MoveL Offs(p0,48.4696,297.2024, 0), v100, z5, tool0;
MoveL Offs(p0,48.6625,297.275, 0), v100, z5, tool0;
MoveL Offs(p0,48.848800000000004,297.9032, 0), v100, z5, tool0;
MoveL Offs(p0,48.7981,298.2614, 0), v100, z5, tool0;
MoveL Offs(p0,48.7,298.7, 0), v100, z5, tool0;
MoveL Offs(p0,48.48880000000001,299.4760000000001, 0), v100, z5, tool0;
MoveL Offs(p0,48.3652,299.978, 0), v100, z5, tool0;
MoveL Offs(p0,48.234399999999994,300.5400000000001, 0), v100, z5, tool0;
MoveL Offs(p0,48.1,301.15, 0), v100, z5, tool0;
MoveL Offs(p0,47.965599999999995,301.796, 0), v100, z5, tool0;
MoveL Offs(p0,47.834799999999994,302.466, 0), v100, z5, tool0;
MoveL Offs(p0,47.711200000000005,303.148, 0), v100, z5, tool0;
MoveL Offs(p0,47.598400000000005,303.83000000000004, 0), v100, z5, tool0;
MoveL Offs(p0,47.5,304.5, 0), v100, z5, tool0;
MoveL Offs(p0,47.17200000000001,306.3952000000001, 0), v100, z5, tool0;
MoveL Offs(p0,47.086,307.0218, 0), v100, z5, tool0;
MoveL Offs(p0,47.06000000000001,307.4456, 0), v100, z5, tool0;
MoveL Offs(p0,47.1,307.675, 0), v100, z5, tool0;
MoveL Offs(p0,47.211999999999996,307.7184, 0), v100, z5, tool0;
MoveL Offs(p0,48.040000000000006,306.8166, 0), v100, z5, tool0;
MoveL Offs(p0,48.5,306.2, 0), v100, z5, tool0;
MoveL Offs(p0,48.75480000000001,305.8350000000001, 0), v100, z5, tool0;
MoveL Offs(p0,48.97840000000001,305.46400000000006, 0), v100, z5, tool0;
MoveL Offs(p0,49.169599999999996,305.09299999999996, 0), v100, z5, tool0;
MoveL Offs(p0,49.3272,304.728, 0), v100, z5, tool0;
MoveL Offs(p0,49.45,304.375, 0), v100, z5, tool0;
MoveL Offs(p0,49.53680000000001,304.04, 0), v100, z5, tool0;
MoveL Offs(p0,49.586400000000005,303.729, 0), v100, z5, tool0;
MoveL Offs(p0,49.5976,303.44800000000004, 0), v100, z5, tool0;
MoveL Offs(p0,49.5692,303.20300000000003, 0), v100, z5, tool0;
MoveL Offs(p0,49.5,303.0, 0), v100, z5, tool0;
MoveL Offs(p0,49.5,303.0, 0), v100, z5, tool0;
MoveJ Offs(p0,394.7,303.0, 10), v100, z1, tool0;
MoveL Offs(p0,393.5853000000001,301.9654, 0), v100, z5, tool0;
MoveL Offs(p0,392.4784000000001,300.6392000000001, 0), v100, z5, tool0;
MoveL Offs(p0,391.4051,299.07779999999997, 0), v100, z5, tool0;
MoveL Offs(p0,390.3912,297.3376, 0), v100, z5, tool0;
MoveL Offs(p0,389.4625,295.475, 0), v100, z5, tool0;
MoveL Offs(p0,388.6448,293.5464, 0), v100, z5, tool0;
MoveL Offs(p0,387.9639,291.6082, 0), v100, z5, tool0;
MoveL Offs(p0,387.4456,289.71680000000003, 0), v100, z5, tool0;
MoveL Offs(p0,387.1157,287.9286, 0), v100, z5, tool0;
MoveL Offs(p0,387.0,286.3, 0), v100, z5, tool0;
MoveL Offs(p0,387.2152000000001,283.32400000000007, 0), v100, z5, tool0;
MoveL Offs(p0,387.4968,281.96200000000005, 0), v100, z5, tool0;
MoveL Offs(p0,387.90560000000005,280.65999999999997, 0), v100, z5, tool0;
MoveL Offs(p0,388.45,279.4, 0), v100, z5, tool0;
MoveL Offs(p0,389.1384,278.164, 0), v100, z5, tool0;
MoveL Offs(p0,389.9792,276.934, 0), v100, z5, tool0;
MoveL Offs(p0,390.9808,275.692, 0), v100, z5, tool0;
MoveL Offs(p0,392.15160000000003,274.42, 0), v100, z5, tool0;
MoveL Offs(p0,393.5,273.1, 0), v100, z5, tool0;
MoveL Offs(p0,394.37790000000007,272.2835000000001, 0), v100, z5, tool0;
MoveL Offs(p0,395.0992000000001,271.56000000000006, 0), v100, z5, tool0;
MoveL Offs(p0,395.6753,270.90849999999995, 0), v100, z5, tool0;
MoveL Offs(p0,396.11760000000004,270.30800000000005, 0), v100, z5, tool0;
MoveL Offs(p0,396.4375,269.7375, 0), v100, z5, tool0;
MoveL Offs(p0,396.64639999999997,269.176, 0), v100, z5, tool0;
MoveL Offs(p0,396.7557,268.6025, 0), v100, z5, tool0;
MoveL Offs(p0,396.77680000000004,267.996, 0), v100, z5, tool0;
MoveL Offs(p0,396.72110000000004,267.3355, 0), v100, z5, tool0;
MoveL Offs(p0,396.6,266.6, 0), v100, z5, tool0;
MoveL Offs(p0,396.2397,265.0522, 0), v100, z5, tool0;
MoveL Offs(p0,395.7936000000001,263.8056000000001, 0), v100, z5, tool0;
MoveL Offs(p0,395.1338999999999,262.8254, 0), v100, z5, tool0;
MoveL Offs(p0,394.13280000000003,262.0768, 0), v100, z5, tool0;
MoveL Offs(p0,392.6625,261.525, 0), v100, z5, tool0;
MoveL Offs(p0,390.59520000000003,261.1352, 0), v100, z5, tool0;
MoveL Offs(p0,387.8031,260.87260000000003, 0), v100, z5, tool0;
MoveL Offs(p0,384.1584,260.7024, 0), v100, z5, tool0;
MoveL Offs(p0,379.5333,260.5898, 0), v100, z5, tool0;
MoveL Offs(p0,373.8,260.5, 0), v100, z5, tool0;
MoveL Offs(p0,359.3056,260.172, 0), v100, z5, tool0;
MoveL Offs(p0,356.8625,260.0, 0), v100, z5, tool0;
MoveL Offs(p0,354.7344,259.78000000000003, 0), v100, z5, tool0;
MoveL Offs(p0,352.8427,259.506, 0), v100, z5, tool0;
MoveL Offs(p0,351.10880000000003,259.172, 0), v100, z5, tool0;
MoveL Offs(p0,349.45410000000004,258.77200000000005, 0), v100, z5, tool0;
MoveL Offs(p0,347.8,258.3, 0), v100, z5, tool0;
MoveL Offs(p0,346.68620000000004,257.98850000000004, 0), v100, z5, tool0;
MoveL Offs(p0,345.6336000000001,257.71600000000007, 0), v100, z5, tool0;
MoveL Offs(p0,344.6554,257.4855, 0), v100, z5, tool0;
MoveL Offs(p0,343.76480000000004,257.3, 0), v100, z5, tool0;
MoveL Offs(p0,342.975,257.1625, 0), v100, z5, tool0;
MoveL Offs(p0,342.2992,257.076, 0), v100, z5, tool0;
MoveL Offs(p0,341.7506,257.0435, 0), v100, z5, tool0;
MoveL Offs(p0,341.34240000000005,257.06800000000004, 0), v100, z5, tool0;
MoveL Offs(p0,341.0878,257.15250000000003, 0), v100, z5, tool0;
MoveL Offs(p0,341.0,257.3, 0), v100, z5, tool0;
MoveL Offs(p0,341.26160000000016,258.04080000000005, 0), v100, z5, tool0;
MoveL Offs(p0,341.57239999999996,258.7112, 0), v100, z5, tool0;
MoveL Offs(p0,341.9888,259.5544, 0), v100, z5, tool0;
MoveL Offs(p0,342.5,260.55, 0), v100, z5, tool0;
MoveL Offs(p0,343.0952,261.6776, 0), v100, z5, tool0;
MoveL Offs(p0,343.76359999999994,262.91679999999997, 0), v100, z5, tool0;
MoveL Offs(p0,344.49440000000004,264.2472000000001, 0), v100, z5, tool0;
MoveL Offs(p0,345.2768,265.64840000000004, 0), v100, z5, tool0;
MoveL Offs(p0,346.1,267.1, 0), v100, z5, tool0;
MoveL Offs(p0,347.2601000000001,269.11800000000005, 0), v100, z5, tool0;
MoveL Offs(p0,348.22880000000015,270.87200000000007, 0), v100, z5, tool0;
MoveL Offs(p0,349.0187,272.392, 0), v100, z5, tool0;
MoveL Offs(p0,349.64240000000007,273.70799999999997, 0), v100, z5, tool0;
MoveL Offs(p0,350.1125,274.85, 0), v100, z5, tool0;
MoveL Offs(p0,350.4416,275.848, 0), v100, z5, tool0;
MoveL Offs(p0,350.6423,276.732, 0), v100, z5, tool0;
MoveL Offs(p0,350.7272,277.53200000000004, 0), v100, z5, tool0;
MoveL Offs(p0,350.70889999999997,278.278, 0), v100, z5, tool0;
MoveL Offs(p0,350.6,279.0, 0), v100, z5, tool0;
MoveL Offs(p0,350.9,282.1, 0), v100, z5, tool0;
MoveL Offs(p0,351.32,282.6504, 0), v100, z5, tool0;
MoveL Offs(p0,351.902,283.2392, 0), v100, z5, tool0;
MoveL Offs(p0,352.66400000000004,283.8928, 0), v100, z5, tool0;
MoveL Offs(p0,353.62399999999997,284.63759999999996, 0), v100, z5, tool0;
MoveL Offs(p0,354.8,285.5, 0), v100, z5, tool0;
MoveL Offs(p0,356.8775,286.9497, 0), v100, z5, tool0;
MoveL Offs(p0,359.34800000000007,288.5176, 0), v100, z5, tool0;
MoveL Offs(p0,362.14849999999996,290.1719, 0), v100, z5, tool0;
MoveL Offs(p0,365.216,291.8808, 0), v100, z5, tool0;
MoveL Offs(p0,368.4875,293.6125, 0), v100, z5, tool0;
MoveL Offs(p0,371.9,295.3352, 0), v100, z5, tool0;
MoveL Offs(p0,375.3905,297.0171, 0), v100, z5, tool0;
MoveL Offs(p0,378.896,298.6264, 0), v100, z5, tool0;
MoveL Offs(p0,382.3535,300.1313, 0), v100, z5, tool0;
MoveL Offs(p0,385.7,301.5, 0), v100, z5, tool0;
MoveL Offs(p0,388.5062000000001,302.5680000000001, 0), v100, z5, tool0;
MoveL Offs(p0,390.8696000000001,303.4320000000001, 0), v100, z5, tool0;
MoveL Offs(p0,392.7974,304.092, 0), v100, z5, tool0;
MoveL Offs(p0,394.29679999999996,304.54800000000006, 0), v100, z5, tool0;
MoveL Offs(p0,395.375,304.8, 0), v100, z5, tool0;
MoveL Offs(p0,396.0392,304.84800000000007, 0), v100, z5, tool0;
MoveL Offs(p0,396.2966,304.692, 0), v100, z5, tool0;
MoveL Offs(p0,396.1544,304.332, 0), v100, z5, tool0;
MoveL Offs(p0,395.61980000000005,303.76800000000003, 0), v100, z5, tool0;
MoveL Offs(p0,394.7,303.0, 0), v100, z5, tool0;
MoveL Offs(p0,394.7,303.0, 0), v100, z5, tool0;
MoveJ Offs(p0,22.5,271.1, 10), v100, z1, tool0;
MoveL Offs(p0,23.33780000000001,268.8337, 0), v100, z5, tool0;
MoveL Offs(p0,24.18640000000001,266.6856000000001, 0), v100, z5, tool0;
MoveL Offs(p0,25.068599999999996,264.6119, 0), v100, z5, tool0;
MoveL Offs(p0,26.0072,262.5688, 0), v100, z5, tool0;
MoveL Offs(p0,27.025,260.5125, 0), v100, z5, tool0;
MoveL Offs(p0,28.144799999999996,258.39919999999995, 0), v100, z5, tool0;
MoveL Offs(p0,29.389400000000002,256.1851, 0), v100, z5, tool0;
MoveL Offs(p0,30.781600000000005,253.8264, 0), v100, z5, tool0;
MoveL Offs(p0,32.3442,251.2793, 0), v100, z5, tool0;
MoveL Offs(p0,34.1,248.5, 0), v100, z5, tool0;
MoveL Offs(p0,34.850500000000004,247.28090000000003, 0), v100, z5, tool0;
MoveL Offs(p0,35.48400000000001,246.19920000000008, 0), v100, z5, tool0;
MoveL Offs(p0,36.003499999999995,245.24829999999997, 0), v100, z5, tool0;
MoveL Offs(p0,36.412,244.42160000000004, 0), v100, z5, tool0;
MoveL Offs(p0,36.7125,243.7125, 0), v100, z5, tool0;
MoveL Offs(p0,36.908,243.1144, 0), v100, z5, tool0;
MoveL Offs(p0,37.0015,242.62070000000003, 0), v100, z5, tool0;
MoveL Offs(p0,36.996,242.22480000000004, 0), v100, z5, tool0;
MoveL Offs(p0,36.8945,241.9201, 0), v100, z5, tool0;
MoveL Offs(p0,36.7,241.7, 0), v100, z5, tool0;
MoveL Offs(p0,36.42160000000001,241.45840000000007, 0), v100, z5, tool0;
MoveL Offs(p0,36.3859,241.37959999999998, 0), v100, z5, tool0;
MoveL Offs(p0,36.41680000000001,241.3272, 0), v100, z5, tool0;
MoveL Offs(p0,37.17040000000001,241.3576, 0), v100, z5, tool0;
MoveL Offs(p0,37.5073,241.4192, 0), v100, z5, tool0;
MoveL Offs(p0,37.9,241.5, 0), v100, z5, tool0;
MoveL Offs(p0,38.72960000000001,241.7272000000001, 0), v100, z5, tool0;
MoveL Offs(p0,39.0484,241.7853, 0), v100, z5, tool0;
MoveL Offs(p0,39.30480000000001,241.8056, 0), v100, z5, tool0;
MoveL Offs(p0,39.5,241.7875, 0), v100, z5, tool0;
MoveL Offs(p0,39.635200000000005,241.7304, 0), v100, z5, tool0;
MoveL Offs(p0,39.6,241.1, 0), v100, z5, tool0;
MoveL Offs(p0,39.3993,240.57799999999997, 0), v100, z5, tool0;
MoveL Offs(p0,39.905100000000004,240.18200000000002, 0), v100, z5, tool0;
MoveL Offs(p0,40.1,240.2, 0), v100, z5, tool0;
MoveL Offs(p0,40.9136,239.93179999999998, 0), v100, z5, tool0;
MoveL Offs(p0,41.24720000000001,239.66559999999998, 0), v100, z5, tool0;
MoveL Offs(p0,41.6,239.325, 0), v100, z5, tool0;
MoveL Offs(p0,41.9648,238.91840000000002, 0), v100, z5, tool0;
MoveL Offs(p0,42.3344,238.4542, 0), v100, z5, tool0;
MoveL Offs(p0,42.701600000000006,237.94080000000002, 0), v100, z5, tool0;
MoveL Offs(p0,43.0592,237.3866, 0), v100, z5, tool0;
MoveL Offs(p0,43.4,236.8, 0), v100, z5, tool0;
MoveL Offs(p0,43.838300000000004,235.98240000000004, 0), v100, z5, tool0;
MoveL Offs(p0,44.19440000000001,235.2632000000001, 0), v100, z5, tool0;
MoveL Offs(p0,44.470099999999995,234.6328, 0), v100, z5, tool0;
MoveL Offs(p0,44.66720000000001,234.08160000000004, 0), v100, z5, tool0;
MoveL Offs(p0,44.7875,233.6, 0), v100, z5, tool0;
MoveL Offs(p0,44.832800000000006,233.17839999999995, 0), v100, z5, tool0;
MoveL Offs(p0,44.804899999999996,232.80720000000002, 0), v100, z5, tool0;
MoveL Offs(p0,44.705600000000004,232.4768, 0), v100, z5, tool0;
MoveL Offs(p0,44.5367,232.17759999999998, 0), v100, z5, tool0;
MoveL Offs(p0,44.3,231.9, 0), v100, z5, tool0;
MoveL Offs(p0,44.02900000000001,231.66020000000003, 0), v100, z5, tool0;
MoveL Offs(p0,43.75200000000001,231.48160000000007, 0), v100, z5, tool0;
MoveL Offs(p0,43.463,231.3654, 0), v100, z5, tool0;
MoveL Offs(p0,43.156000000000006,231.3128, 0), v100, z5, tool0;
MoveL Offs(p0,42.825,231.325, 0), v100, z5, tool0;
MoveL Offs(p0,42.464,231.40320000000003, 0), v100, z5, tool0;
MoveL Offs(p0,42.067,231.5486, 0), v100, z5, tool0;
MoveL Offs(p0,40.6,232.4, 0), v100, z5, tool0;
MoveL Offs(p0,40.16270000000001,232.67810000000003, 0), v100, z5, tool0;
MoveL Offs(p0,39.75360000000001,232.96880000000004, 0), v100, z5, tool0;
MoveL Offs(p0,39.37689999999999,233.2667, 0), v100, z5, tool0;
MoveL Offs(p0,39.0368,233.56640000000002, 0), v100, z5, tool0;
MoveL Offs(p0,38.7375,233.8625, 0), v100, z5, tool0;
MoveL Offs(p0,38.4832,234.14960000000002, 0), v100, z5, tool0;
MoveL Offs(p0,38.2781,234.4223, 0), v100, z5, tool0;
MoveL Offs(p0,38.126400000000004,234.67520000000005, 0), v100, z5, tool0;
MoveL Offs(p0,38.032300000000006,234.9029, 0), v100, z5, tool0;
MoveL Offs(p0,38.0,235.1, 0), v100, z5, tool0;
MoveL Offs(p0,37.751599999999996,235.95049999999998, 0), v100, z5, tool0;
MoveL Offs(p0,37.5712,236.348, 0), v100, z5, tool0;
MoveL Offs(p0,37.35,236.7875, 0), v100, z5, tool0;
MoveL Offs(p0,37.0928,237.26, 0), v100, z5, tool0;
MoveL Offs(p0,36.8044,237.75650000000002, 0), v100, z5, tool0;
MoveL Offs(p0,36.48960000000001,238.26800000000003, 0), v100, z5, tool0;
MoveL Offs(p0,36.153200000000005,238.78550000000004, 0), v100, z5, tool0;
MoveL Offs(p0,35.8,239.3, 0), v100, z5, tool0;
MoveL Offs(p0,34.16930000000001,241.69430000000006, 0), v100, z5, tool0;
MoveL Offs(p0,32.39040000000001,244.57040000000006, 0), v100, z5, tool0;
MoveL Offs(p0,30.5431,247.7681, 0), v100, z5, tool0;
MoveL Offs(p0,28.7072,251.12720000000004, 0), v100, z5, tool0;
MoveL Offs(p0,26.9625,254.4875, 0), v100, z5, tool0;
MoveL Offs(p0,25.388799999999996,257.6888, 0), v100, z5, tool0;
MoveL Offs(p0,24.0659,260.5709, 0), v100, z5, tool0;
MoveL Offs(p0,23.073600000000003,262.9736, 0), v100, z5, tool0;
MoveL Offs(p0,22.4917,264.73670000000004, 0), v100, z5, tool0;
MoveL Offs(p0,22.4,265.7, 0), v100, z5, tool0;
MoveL Offs(p0,22.2,267.0, 0), v100, z5, tool0;
MoveL Offs(p0,21.6107,267.5379, 0), v100, z5, tool0;
MoveL Offs(p0,20.89360000000001,269.02320000000003, 0), v100, z5, tool0;
MoveL Offs(p0,20.094900000000003,271.26329999999996, 0), v100, z5, tool0;
MoveL Offs(p0,19.2608,274.0656, 0), v100, z5, tool0;
MoveL Offs(p0,18.4375,277.2375, 0), v100, z5, tool0;
MoveL Offs(p0,17.6712,280.5864, 0), v100, z5, tool0;
MoveL Offs(p0,17.0081,283.9197, 0), v100, z5, tool0;
MoveL Offs(p0,16.494400000000002,287.0448, 0), v100, z5, tool0;
MoveL Offs(p0,16.1763,289.76910000000004, 0), v100, z5, tool0;
MoveL Offs(p0,16.1,291.9, 0), v100, z5, tool0;
MoveL Offs(p0,16.3214,292.1826, 0), v100, z5, tool0;
MoveL Offs(p0,16.675,291.375, 0), v100, z5, tool0;
MoveL Offs(p0,16.8992,290.7048, 0), v100, z5, tool0;
MoveL Offs(p0,17.1486,289.8714, 0), v100, z5, tool0;
MoveL Offs(p0,17.418400000000002,288.8856, 0), v100, z5, tool0;
MoveL Offs(p0,17.7038,287.75820000000004, 0), v100, z5, tool0;
MoveL Offs(p0,18.0,286.5, 0), v100, z5, tool0;
MoveL Offs(p0,18.328500000000005,285.11030000000005, 0), v100, z5, tool0;
MoveL Offs(p0,18.708000000000006,283.6024000000001, 0), v100, z5, tool0;
MoveL Offs(p0,19.1295,282.00809999999996, 0), v100, z5, tool0;
MoveL Offs(p0,19.584,280.3592, 0), v100, z5, tool0;
MoveL Offs(p0,20.0625,278.6875, 0), v100, z5, tool0;
MoveL Offs(p0,20.556,277.02479999999997, 0), v100, z5, tool0;
MoveL Offs(p0,21.055500000000002,275.4029, 0), v100, z5, tool0;
MoveL Offs(p0,21.552000000000003,273.85360000000003, 0), v100, z5, tool0;
MoveL Offs(p0,22.0365,272.4087, 0), v100, z5, tool0;
MoveL Offs(p0,22.5,271.1, 0), v100, z5, tool0;
MoveL Offs(p0,22.5,271.1, 0), v100, z5, tool0;
MoveJ Offs(p0,36.1,288.1, 10), v100, z1, tool0;
MoveL Offs(p0,36.39620000000001,288.49760000000003, 0), v100, z5, tool0;
MoveL Offs(p0,36.68160000000002,288.9048000000001, 0), v100, z5, tool0;
MoveL Offs(p0,36.95139999999999,289.3132, 0), v100, z5, tool0;
MoveL Offs(p0,37.2008,289.71439999999996, 0), v100, z5, tool0;
MoveL Offs(p0,37.425,290.1, 0), v100, z5, tool0;
MoveL Offs(p0,37.6192,290.4616, 0), v100, z5, tool0;
MoveL Offs(p0,37.7786,290.7908, 0), v100, z5, tool0;
MoveL Offs(p0,37.8984,291.0792, 0), v100, z5, tool0;
MoveL Offs(p0,37.973800000000004,291.3184, 0), v100, z5, tool0;
MoveL Offs(p0,38.0,291.5, 0), v100, z5, tool0;
MoveL Offs(p0,38.6875,291.0625, 0), v100, z5, tool0;
MoveL Offs(p0,38.93599999999999,290.70079999999996, 0), v100, z5, tool0;
MoveL Offs(p0,39.2145,290.2659, 0), v100, z5, tool0;
MoveL Offs(p0,39.52,289.7656, 0), v100, z5, tool0;
MoveL Offs(p0,39.8495,289.20770000000005, 0), v100, z5, tool0;
MoveL Offs(p0,40.2,288.6, 0), v100, z5, tool0;
MoveL Offs(p0,42.2,284.6, 0), v100, z5, tool0;
MoveL Offs(p0,44.0,286.9, 0), v100, z5, tool0;
MoveL Offs(p0,44.4371,287.49449999999996, 0), v100, z5, tool0;
MoveL Offs(p0,44.79680000000001,287.9600000000001, 0), v100, z5, tool0;
MoveL Offs(p0,45.0917,288.29949999999997, 0), v100, z5, tool0;
MoveL Offs(p0,45.3344,288.516, 0), v100, z5, tool0;
MoveL Offs(p0,45.5375,288.6125, 0), v100, z5, tool0;
MoveL Offs(p0,45.7136,288.592, 0), v100, z5, tool0;
MoveL Offs(p0,45.8753,288.4575, 0), v100, z5, tool0;
MoveL Offs(p0,46.03520000000001,288.212, 0), v100, z5, tool0;
MoveL Offs(p0,46.2059,287.8585, 0), v100, z5, tool0;
MoveL Offs(p0,46.4,287.4, 0), v100, z5, tool0;
MoveL Offs(p0,46.998400000000004,284.9322, 0), v100, z5, tool0;
MoveL Offs(p0,47.41920000000002,281.10960000000006, 0), v100, z5, tool0;
MoveL Offs(p0,47.6708,276.2634, 0), v100, z5, tool0;
MoveL Offs(p0,47.7616,270.7248, 0), v100, z5, tool0;
MoveL Offs(p0,47.7,264.825, 0), v100, z5, tool0;
MoveL Offs(p0,47.4944,258.89520000000005, 0), v100, z5, tool0;
MoveL Offs(p0,47.1532,253.2666, 0), v100, z5, tool0;
MoveL Offs(p0,46.68480000000001,248.27040000000002, 0), v100, z5, tool0;
MoveL Offs(p0,46.0976,244.23780000000002, 0), v100, z5, tool0;
MoveL Offs(p0,45.4,241.5, 0), v100, z5, tool0;
MoveL Offs(p0,44.52810000000001,240.81270000000004, 0), v100, z5, tool0;
MoveL Offs(p0,41.1367,243.1029, 0), v100, z5, tool0;
MoveL Offs(p0,38.8464,245.75280000000004, 0), v100, z5, tool0;
MoveL Offs(p0,36.3125,249.1875, 0), v100, z5, tool0;
MoveL Offs(p0,33.6496,253.24319999999997, 0), v100, z5, tool0;
MoveL Offs(p0,30.972299999999997,257.7561, 0), v100, z5, tool0;
MoveL Offs(p0,28.3952,262.5624, 0), v100, z5, tool0;
MoveL Offs(p0,26.0329,267.49830000000003, 0), v100, z5, tool0;
MoveL Offs(p0,24.0,272.4, 0), v100, z5, tool0;
MoveL Offs(p0,23.035600000000002,275.0069000000001, 0), v100, z5, tool0;
MoveL Offs(p0,22.188800000000004,277.5712000000001, 0), v100, z5, tool0;
MoveL Offs(p0,21.4692,280.0383, 0), v100, z5, tool0;
MoveL Offs(p0,20.886400000000002,282.3536, 0), v100, z5, tool0;
MoveL Offs(p0,20.45,284.4625, 0), v100, z5, tool0;
MoveL Offs(p0,20.1696,286.3104, 0), v100, z5, tool0;
MoveL Offs(p0,20.0548,287.84270000000004, 0), v100, z5, tool0;
MoveL Offs(p0,20.115200000000005,289.00480000000005, 0), v100, z5, tool0;
MoveL Offs(p0,20.3604,289.74210000000005, 0), v100, z5, tool0;
MoveL Offs(p0,20.8,290.0, 0), v100, z5, tool0;
MoveL Offs(p0,21.5047,289.703, 0), v100, z5, tool0;
MoveL Offs(p0,21.7984,289.48800000000006, 0), v100, z5, tool0;
MoveL Offs(p0,22.1125,289.225, 0), v100, z5, tool0;
MoveL Offs(p0,22.4416,288.91999999999996, 0), v100, z5, tool0;
MoveL Offs(p0,22.7803,288.579, 0), v100, z5, tool0;
MoveL Offs(p0,23.123200000000004,288.20799999999997, 0), v100, z5, tool0;
MoveL Offs(p0,23.4649,287.813, 0), v100, z5, tool0;
MoveL Offs(p0,23.8,287.4, 0), v100, z5, tool0;
MoveL Offs(p0,25.7,284.7, 0), v100, z5, tool0;
MoveL Offs(p0,28.0,288.4, 0), v100, z5, tool0;
MoveL Offs(p0,30.2,292.1, 0), v100, z5, tool0;
MoveL Offs(p0,32.2,288.9, 0), v100, z5, tool0;
MoveL Offs(p0,34.2,285.6, 0), v100, z5, tool0;
MoveL Offs(p0,36.1,288.1, 0), v100, z5, tool0;
MoveL Offs(p0,36.1,288.1, 0), v100, z5, tool0;
MoveJ Offs(p0,86.6,282.4, 10), v100, z1, tool0;
MoveL Offs(p0,86.38880000000003,279.65520000000004, 0), v100, z5, tool0;
MoveL Offs(p0,86.26520000000001,278.3698, 0), v100, z5, tool0;
MoveL Offs(p0,86.13440000000001,277.1696, 0), v100, z5, tool0;
MoveL Offs(p0,86.0,276.075, 0), v100, z5, tool0;
MoveL Offs(p0,85.8656,275.1064, 0), v100, z5, tool0;
MoveL Offs(p0,85.73479999999999,274.28419999999994, 0), v100, z5, tool0;
MoveL Offs(p0,85.61120000000001,273.62880000000007, 0), v100, z5, tool0;
MoveL Offs(p0,85.49839999999999,273.16060000000004, 0), v100, z5, tool0;
MoveL Offs(p0,85.4,272.9, 0), v100, z5, tool0;
MoveL Offs(p0,85.0895,272.0855, 0), v100, z5, tool0;
MoveL Offs(p0,84.976,271.676, 0), v100, z5, tool0;
MoveL Offs(p0,84.8625,271.2125, 0), v100, z5, tool0;
MoveL Offs(p0,84.752,270.70399999999995, 0), v100, z5, tool0;
MoveL Offs(p0,84.64750000000001,270.1595, 0), v100, z5, tool0;
MoveL Offs(p0,84.552,269.588, 0), v100, z5, tool0;
MoveL Offs(p0,84.4685,268.99850000000004, 0), v100, z5, tool0;
MoveL Offs(p0,84.4,268.4, 0), v100, z5, tool0;
MoveL Offs(p0,83.85910000000001,265.5085, 0), v100, z5, tool0;
MoveL Offs(p0,82.94080000000002,262.04400000000004, 0), v100, z5, tool0;
MoveL Offs(p0,81.71169999999998,258.1715, 0), v100, z5, tool0;
MoveL Offs(p0,80.2384,254.05599999999998, 0), v100, z5, tool0;
MoveL Offs(p0,78.5875,249.8625, 0), v100, z5, tool0;
MoveL Offs(p0,76.8256,245.756, 0), v100, z5, tool0;
MoveL Offs(p0,75.0193,241.9015, 0), v100, z5, tool0;
MoveL Offs(p0,73.2352,238.46400000000003, 0), v100, z5, tool0;
MoveL Offs(p0,71.5399,235.6085, 0), v100, z5, tool0;
MoveL Offs(p0,70.0,233.5, 0), v100, z5, tool0;
MoveL Offs(p0,69.5334,232.9835, 0), v100, z5, tool0;
MoveL Offs(p0,69.03920000000002,232.40400000000008, 0), v100, z5, tool0;
MoveL Offs(p0,68.52579999999999,231.7765, 0), v100, z5, tool0;
MoveL Offs(p0,68.00160000000001,231.11600000000004, 0), v100, z5, tool0;
MoveL Offs(p0,67.475,230.4375, 0), v100, z5, tool0;
MoveL Offs(p0,66.95439999999999,229.756, 0), v100, z5, tool0;
MoveL Offs(p0,66.4482,229.08649999999997, 0), v100, z5, tool0;
MoveL Offs(p0,65.9648,228.44400000000005, 0), v100, z5, tool0;
MoveL Offs(p0,65.51259999999999,227.84350000000003, 0), v100, z5, tool0;
MoveL Offs(p0,65.1,227.3, 0), v100, z5, tool0;
MoveL Offs(p0,64.72650000000002,226.77020000000002, 0), v100, z5, tool0;
MoveL Offs(p0,64.33200000000001,226.2656000000001, 0), v100, z5, tool0;
MoveL Offs(p0,63.9255,225.79339999999996, 0), v100, z5, tool0;
MoveL Offs(p0,63.516000000000005,225.3608, 0), v100, z5, tool0;
MoveL Offs(p0,63.1125,224.975, 0), v100, z5, tool0;
MoveL Offs(p0,62.724000000000004,224.64319999999998, 0), v100, z5, tool0;
MoveL Offs(p0,62.359500000000004,224.3726, 0), v100, z5, tool0;
MoveL Offs(p0,62.028,224.17040000000003, 0), v100, z5, tool0;
MoveL Offs(p0,61.7385,224.0438, 0), v100, z5, tool0;
MoveL Offs(p0,61.5,224.0, 0), v100, z5, tool0;
MoveL Offs(p0,60.981700000000004,224.25660000000002, 0), v100, z5, tool0;
MoveL Offs(p0,60.78560000000001,224.97280000000006, 0), v100, z5, tool0;
MoveL Offs(p0,60.8799,226.0682, 0), v100, z5, tool0;
MoveL Offs(p0,61.23280000000001,227.46239999999997, 0), v100, z5, tool0;
MoveL Offs(p0,61.8125,229.075, 0), v100, z5, tool0;
MoveL Offs(p0,62.58720000000001,230.82559999999998, 0), v100, z5, tool0;
MoveL Offs(p0,63.525099999999995,232.6338, 0), v100, z5, tool0;
MoveL Offs(p0,64.59440000000001,234.4192, 0), v100, z5, tool0;
MoveL Offs(p0,65.7633,236.1014, 0), v100, z5, tool0;
MoveL Offs(p0,67.0,237.6, 0), v100, z5, tool0;
MoveL Offs(p0,67.62470000000002,238.30800000000005, 0), v100, z5, tool0;
MoveL Offs(p0,68.28960000000002,239.10000000000014, 0), v100, z5, tool0;
MoveL Offs(p0,68.98089999999999,239.958, 0), v100, z5, tool0;
MoveL Offs(p0,69.68480000000001,240.86400000000003, 0), v100, z5, tool0;
MoveL Offs(p0,70.3875,241.8, 0), v100, z5, tool0;
MoveL Offs(p0,71.0752,242.74799999999996, 0), v100, z5, tool0;
MoveL Offs(p0,71.7341,243.69, 0), v100, z5, tool0;
MoveL Offs(p0,72.35040000000001,244.608, 0), v100, z5, tool0;
MoveL Offs(p0,72.91029999999999,245.484, 0), v100, z5, tool0;
MoveL Offs(p0,73.4,246.3, 0), v100, z5, tool0;
MoveL Offs(p0,74.3298,247.97310000000007, 0), v100, z5, tool0;
MoveL Offs(p0,75.45040000000003,250.1808000000001, 0), v100, z5, tool0;
MoveL Offs(p0,76.6886,252.7557, 0), v100, z5, tool0;
MoveL Offs(p0,77.9712,255.53040000000001, 0), v100, z5, tool0;
MoveL Offs(p0,79.225,258.3375, 0), v100, z5, tool0;
MoveL Offs(p0,80.3768,261.0096, 0), v100, z5, tool0;
MoveL Offs(p0,81.35340000000001,263.37929999999994, 0), v100, z5, tool0;
MoveL Offs(p0,82.08160000000001,265.27920000000006, 0), v100, z5, tool0;
MoveL Offs(p0,82.4882,266.54190000000006, 0), v100, z5, tool0;
MoveL Offs(p0,82.5,267.0, 0), v100, z5, tool0;
MoveL Offs(p0,82.7121,268.7934, 0), v100, z5, tool0;
MoveL Offs(p0,82.8264,269.2656, 0), v100, z5, tool0;
MoveL Offs(p0,82.95630000000001,269.77020000000005, 0), v100, z5, tool0;
MoveL Offs(p0,83.1,270.3, 0), v100, z5, tool0;
MoveL Offs(p0,83.40750000000001,271.3081, 0), v100, z5, tool0;
MoveL Offs(p0,83.67600000000002,272.26880000000006, 0), v100, z5, tool0;
MoveL Offs(p0,83.9145,273.23670000000004, 0), v100, z5, tool0;
MoveL Offs(p0,84.132,274.2664, 0), v100, z5, tool0;
MoveL Offs(p0,84.3375,275.4125, 0), v100, z5, tool0;
MoveL Offs(p0,84.53999999999999,276.7296, 0), v100, z5, tool0;
MoveL Offs(p0,84.74849999999999,278.2723, 0), v100, z5, tool0;
MoveL Offs(p0,84.97200000000001,280.09520000000003, 0), v100, z5, tool0;
MoveL Offs(p0,85.21950000000001,282.25290000000007, 0), v100, z5, tool0;
MoveL Offs(p0,85.5,284.8, 0), v100, z5, tool0;
MoveL Offs(p0,85.8197,287.23570000000007, 0), v100, z5, tool0;
MoveL Offs(p0,86.11360000000002,289.0336000000001, 0), v100, z5, tool0;
MoveL Offs(p0,86.3739,290.20989999999995, 0), v100, z5, tool0;
MoveL Offs(p0,86.5928,290.7808, 0), v100, z5, tool0;
MoveL Offs(p0,86.7625,290.7625, 0), v100, z5, tool0;
MoveL Offs(p0,86.87519999999999,290.1712, 0), v100, z5, tool0;
MoveL Offs(p0,86.9231,289.0231, 0), v100, z5, tool0;
MoveL Offs(p0,86.89840000000001,287.3344, 0), v100, z5, tool0;
MoveL Offs(p0,86.7933,285.1213, 0), v100, z5, tool0;
MoveL Offs(p0,86.6,282.4, 0), v100, z5, tool0;
MoveL Offs(p0,86.6,282.4, 0), v100, z5, tool0;
MoveJ Offs(p0,149.5,287.9, 10), v100, z1, tool0;
MoveL Offs(p0,149.73039999999997,286.9244, 0), v100, z5, tool0;
MoveL Offs(p0,149.7528,286.58480000000003, 0), v100, z5, tool0;
MoveL Offs(p0,149.75,286.25, 0), v100, z5, tool0;
MoveL Offs(p0,149.7232,285.92719999999997, 0), v100, z5, tool0;
MoveL Offs(p0,149.1777,284.40770000000003, 0), v100, z5, tool0;
MoveL Offs(p0,149.1664,284.30640000000005, 0), v100, z5, tool0;
MoveL Offs(p0,149.1875,284.2375, 0), v100, z5, tool0;
MoveL Offs(p0,149.60790000000003,284.2979, 0), v100, z5, tool0;
MoveL Offs(p0,149.8,284.4, 0), v100, z5, tool0;
MoveL Offs(p0,150.95559999999998,284.1885, 0), v100, z5, tool0;
MoveL Offs(p0,151.1312,283.656, 0), v100, z5, tool0;
MoveL Offs(p0,151.2,282.9375, 0), v100, z5, tool0;
MoveL Offs(p0,151.16079999999997,282.06000000000006, 0), v100, z5, tool0;
MoveL Offs(p0,151.0124,281.0505, 0), v100, z5, tool0;
MoveL Offs(p0,150.7536,279.93600000000004, 0), v100, z5, tool0;
MoveL Offs(p0,150.38320000000002,278.74350000000004, 0), v100, z5, tool0;
MoveL Offs(p0,148.91250000000005,274.55550000000005, 0), v100, z5, tool0;
MoveL Offs(p0,148.16800000000003,270.98400000000004, 0), v100, z5, tool0;
MoveL Offs(p0,147.6635,266.9385, 0), v100, z5, tool0;
MoveL Offs(p0,147.39600000000002,262.572, 0), v100, z5, tool0;
MoveL Offs(p0,147.3625,258.0375, 0), v100, z5, tool0;
MoveL Offs(p0,147.56,253.488, 0), v100, z5, tool0;
MoveL Offs(p0,147.9855,249.07649999999998, 0), v100, z5, tool0;
MoveL Offs(p0,148.63600000000002,244.95600000000005, 0), v100, z5, tool0;
MoveL Offs(p0,149.5085,241.2795, 0), v100, z5, tool0;
MoveL Offs(p0,150.6,238.2, 0), v100, z5, tool0;
MoveL Offs(p0,150.88770000000002,237.59880000000004, 0), v100, z5, tool0;
MoveL Offs(p0,151.14960000000002,237.00240000000002, 0), v100, z5, tool0;
MoveL Offs(p0,151.3839,236.42160000000004, 0), v100, z5, tool0;
MoveL Offs(p0,151.58880000000002,235.86720000000005, 0), v100, z5, tool0;
MoveL Offs(p0,151.7625,235.35, 0), v100, z5, tool0;
MoveL Offs(p0,151.90320000000003,234.8808, 0), v100, z5, tool0;
MoveL Offs(p0,152.0091,234.4704, 0), v100, z5, tool0;
MoveL Offs(p0,152.07840000000002,234.12960000000004, 0), v100, z5, tool0;
MoveL Offs(p0,152.10930000000002,233.8692, 0), v100, z5, tool0;
MoveL Offs(p0,152.1,233.7, 0), v100, z5, tool0;
MoveL Offs(p0,152.3952,233.2536, 0), v100, z5, tool0;
MoveL Offs(p0,152.5221,233.2723, 0), v100, z5, tool0;
MoveL Offs(p0,152.6664,233.3192, 0), v100, z5, tool0;
MoveL Offs(p0,152.8263,233.3949, 0), v100, z5, tool0;
MoveL Offs(p0,153.0,233.5, 0), v100, z5, tool0;
MoveL Offs(p0,153.9855,233.26510000000002, 0), v100, z5, tool0;
MoveL Offs(p0,154.0,233.1, 0), v100, z5, tool0;
MoveL Offs(p0,153.79520000000002,232.78000000000006, 0), v100, z5, tool0;
MoveL Offs(p0,153.55180000000001,232.60950000000003, 0), v100, z5, tool0;
MoveL Offs(p0,153.22560000000001,232.43599999999998, 0), v100, z5, tool0;
MoveL Offs(p0,152.825,232.2625, 0), v100, z5, tool0;
MoveL Offs(p0,152.35840000000002,232.092, 0), v100, z5, tool0;
MoveL Offs(p0,151.8342,231.9275, 0), v100, z5, tool0;
MoveL Offs(p0,151.26080000000002,231.77200000000002, 0), v100, z5, tool0;
MoveL Offs(p0,150.6466,231.62849999999997, 0), v100, z5, tool0;
MoveL Offs(p0,150.0,231.5, 0), v100, z5, tool0;
MoveL Offs(p0,148.71520000000004,231.22800000000007, 0), v100, z5, tool0;
MoveL Offs(p0,148.1118,231.0725, 0), v100, z5, tool0;
MoveL Offs(p0,147.5456,230.90800000000004, 0), v100, z5, tool0;
MoveL Offs(p0,147.025,230.7375, 0), v100, z5, tool0;
MoveL Offs(p0,146.55839999999998,230.564, 0), v100, z5, tool0;
MoveL Offs(p0,146.1542,230.39049999999997, 0), v100, z5, tool0;
MoveL Offs(p0,145.82080000000002,230.21999999999997, 0), v100, z5, tool0;
MoveL Offs(p0,145.56660000000002,230.05550000000002, 0), v100, z5, tool0;
MoveL Offs(p0,145.4,229.9, 0), v100, z5, tool0;
MoveL Offs(p0,145.04210000000003,229.44020000000006, 0), v100, z5, tool0;
MoveL Offs(p0,144.63680000000005,229.13760000000002, 0), v100, z5, tool0;
MoveL Offs(p0,144.19670000000002,228.98740000000004, 0), v100, z5, tool0;
MoveL Offs(p0,143.7344,228.9848, 0), v100, z5, tool0;
MoveL Offs(p0,143.2625,229.125, 0), v100, z5, tool0;
MoveL Offs(p0,142.7936,229.40319999999997, 0), v100, z5, tool0;
MoveL Offs(p0,141.9152,230.3544, 0), v100, z5, tool0;
MoveL Offs(p0,141.53090000000003,231.0178, 0), v100, z5, tool0;
MoveL Offs(p0,141.2,231.8, 0), v100, z5, tool0;
MoveL Offs(p0,139.91450000000003,236.19530000000003, 0), v100, z5, tool0;
MoveL Offs(p0,138.99200000000002,241.48640000000006, 0), v100, z5, tool0;
MoveL Offs(p0,138.4235,247.44109999999995, 0), v100, z5, tool0;
MoveL Offs(p0,138.2,253.8272, 0), v100, z5, tool0;
MoveL Offs(p0,138.3125,260.4125, 0), v100, z5, tool0;
MoveL Offs(p0,138.752,266.9648, 0), v100, z5, tool0;
MoveL Offs(p0,139.5095,273.25190000000003, 0), v100, z5, tool0;
MoveL Offs(p0,140.57600000000002,279.0416, 0), v100, z5, tool0;
MoveL Offs(p0,141.9425,284.1017, 0), v100, z5, tool0;
MoveL Offs(p0,143.6,288.2, 0), v100, z5, tool0;
MoveL Offs(p0,144.127,289.007, 0), v100, z5, tool0;
MoveL Offs(p0,144.73200000000003,289.62800000000004, 0), v100, z5, tool0;
MoveL Offs(p0,145.391,290.063, 0), v100, z5, tool0;
MoveL Offs(p0,146.08,290.312, 0), v100, z5, tool0;
MoveL Offs(p0,146.775,290.375, 0), v100, z5, tool0;
MoveL Offs(p0,147.452,290.25199999999995, 0), v100, z5, tool0;
MoveL Offs(p0,148.087,289.943, 0), v100, z5, tool0;
MoveL Offs(p0,148.656,289.44800000000004, 0), v100, z5, tool0;
MoveL Offs(p0,149.13500000000002,288.767, 0), v100, z5, tool0;
MoveL Offs(p0,149.5,287.9, 0), v100, z5, tool0;
MoveL Offs(p0,149.5,287.9, 0), v100, z5, tool0;
MoveJ Offs(p0,156.2,285.7, 10), v100, z1, tool0;
MoveL Offs(p0,156.5645,282.5032, 0), v100, z5, tool0;
MoveL Offs(p0,156.96,281.3624, 0), v100, z5, tool0;
MoveL Offs(p0,157.4875,280.2, 0), v100, z5, tool0;
MoveL Offs(p0,158.144,279.0256, 0), v100, z5, tool0;
MoveL Offs(p0,158.92649999999998,277.84880000000004, 0), v100, z5, tool0;
MoveL Offs(p0,159.83200000000002,276.67920000000004, 0), v100, z5, tool0;
MoveL Offs(p0,160.85750000000002,275.5264, 0), v100, z5, tool0;
MoveL Offs(p0,162.0,274.4, 0), v100, z5, tool0;
MoveL Offs(p0,162.92490000000004,273.48810000000003, 0), v100, z5, tool0;
MoveL Offs(p0,163.66320000000005,272.72080000000005, 0), v100, z5, tool0;
MoveL Offs(p0,164.2203,272.0806999999999, 0), v100, z5, tool0;
MoveL Offs(p0,164.60160000000002,271.5504, 0), v100, z5, tool0;
MoveL Offs(p0,164.8125,271.1125, 0), v100, z5, tool0;
MoveL Offs(p0,164.8584,270.7496, 0), v100, z5, tool0;
MoveL Offs(p0,164.74470000000002,270.4443, 0), v100, z5, tool0;
MoveL Offs(p0,164.4768,270.17920000000004, 0), v100, z5, tool0;
MoveL Offs(p0,164.0601,269.93690000000004, 0), v100, z5, tool0;
MoveL Offs(p0,163.5,269.7, 0), v100, z5, tool0;
MoveL Offs(p0,161.76479999999998,270.26969999999994, 0), v100, z5, tool0;
MoveL Offs(p0,161.0616,270.8584, 0), v100, z5, tool0;
MoveL Offs(p0,160.35,271.5875, 0), v100, z5, tool0;
MoveL Offs(p0,159.6624,272.4216, 0), v100, z5, tool0;
MoveL Offs(p0,159.03119999999998,273.32529999999997, 0), v100, z5, tool0;
MoveL Offs(p0,158.4888,274.2632, 0), v100, z5, tool0;
MoveL Offs(p0,158.0676,275.19989999999996, 0), v100, z5, tool0;
MoveL Offs(p0,157.8,276.1, 0), v100, z5, tool0;
MoveL Offs(p0,157.57410000000002,276.80649999999997, 0), v100, z5, tool0;
MoveL Offs(p0,157.4832,277.02799999999996, 0), v100, z5, tool0;
MoveL Offs(p0,157.3875,277.2375, 0), v100, z5, tool0;
MoveL Offs(p0,157.2888,277.43199999999996, 0), v100, z5, tool0;
MoveL Offs(p0,157.1889,277.6085, 0), v100, z5, tool0;
MoveL Offs(p0,157.08960000000002,277.764, 0), v100, z5, tool0;
MoveL Offs(p0,156.9927,277.8955, 0), v100, z5, tool0;
MoveL Offs(p0,156.9,278.0, 0), v100, z5, tool0;
MoveL Offs(p0,156.6207,278.41780000000006, 0), v100, z5, tool0;
MoveL Offs(p0,156.22560000000004,279.1944000000001, 0), v100, z5, tool0;
MoveL Offs(p0,155.7489,280.2446, 0), v100, z5, tool0;
MoveL Offs(p0,155.22480000000002,281.4832, 0), v100, z5, tool0;
MoveL Offs(p0,154.6875,282.825, 0), v100, z5, tool0;
MoveL Offs(p0,154.17120000000003,284.1848, 0), v100, z5, tool0;
MoveL Offs(p0,153.71009999999998,285.47740000000005, 0), v100, z5, tool0;
MoveL Offs(p0,153.3384,286.61760000000004, 0), v100, z5, tool0;
MoveL Offs(p0,153.0903,287.52020000000005, 0), v100, z5, tool0;
MoveL Offs(p0,153.0,288.1, 0), v100, z5, tool0;
MoveL Offs(p0,153.34560000000002,288.6632, 0), v100, z5, tool0;
MoveL Offs(p0,153.525,288.75, 0), v100, z5, tool0;
MoveL Offs(p0,153.7344,288.81280000000004, 0), v100, z5, tool0;
MoveL Offs(p0,153.97020000000003,288.8504, 0), v100, z5, tool0;
MoveL Offs(p0,154.2288,288.8616, 0), v100, z5, tool0;
MoveL Offs(p0,154.5066,288.84520000000003, 0), v100, z5, tool0;
MoveL Offs(p0,154.8,288.8, 0), v100, z5, tool0;
MoveL Offs(p0,155.42560000000006,288.5448000000001, 0), v100, z5, tool0;
MoveL Offs(p0,155.6694,288.35720000000003, 0), v100, z5, tool0;
MoveL Offs(p0,155.86880000000002,288.1264, 0), v100, z5, tool0;
MoveL Offs(p0,156.025,287.85, 0), v100, z5, tool0;
MoveL Offs(p0,156.1392,287.52560000000005, 0), v100, z5, tool0;
MoveL Offs(p0,156.2126,287.1508, 0), v100, z5, tool0;
MoveL Offs(p0,156.2464,286.7232, 0), v100, z5, tool0;
MoveL Offs(p0,156.2418,286.2404, 0), v100, z5, tool0;
MoveL Offs(p0,156.2,285.7, 0), v100, z5, tool0;
MoveL Offs(p0,156.2,285.7, 0), v100, z5, tool0;
MoveJ Offs(p0,172.8,284.9, 10), v100, z1, tool0;
MoveL Offs(p0,173.7997,284.68750000000006, 0), v100, z5, tool0;
MoveL Offs(p0,174.74960000000004,284.4720000000001, 0), v100, z5, tool0;
MoveL Offs(p0,175.63590000000002,284.2565, 0), v100, z5, tool0;
MoveL Offs(p0,176.44480000000004,284.044, 0), v100, z5, tool0;
MoveL Offs(p0,177.1625,283.8375, 0), v100, z5, tool0;
MoveL Offs(p0,177.77519999999998,283.64, 0), v100, z5, tool0;
MoveL Offs(p0,178.2691,283.4545, 0), v100, z5, tool0;
MoveL Offs(p0,178.6304,283.284, 0), v100, z5, tool0;
MoveL Offs(p0,178.8453,283.1315, 0), v100, z5, tool0;
MoveL Offs(p0,178.9,283.0, 0), v100, z5, tool0;
MoveL Offs(p0,178.62640000000005,282.6160000000001, 0), v100, z5, tool0;
MoveL Offs(p0,178.30059999999997,282.2845, 0), v100, z5, tool0;
MoveL Offs(p0,177.8632,281.872, 0), v100, z5, tool0;
MoveL Offs(p0,177.325,281.3875, 0), v100, z5, tool0;
MoveL Offs(p0,176.6968,280.84000000000003, 0), v100, z5, tool0;
MoveL Offs(p0,175.9894,280.2385, 0), v100, z5, tool0;
MoveL Offs(p0,175.21359999999999,279.592, 0), v100, z5, tool0;
MoveL Offs(p0,174.3802,278.90950000000004, 0), v100, z5, tool0;
MoveL Offs(p0,173.5,278.2, 0), v100, z5, tool0;
MoveL Offs(p0,171.80930000000004,276.9081, 0), v100, z5, tool0;
MoveL Offs(p0,170.36640000000006,275.9168000000001, 0), v100, z5, tool0;
MoveL Offs(p0,169.1251,275.23269999999997, 0), v100, z5, tool0;
MoveL Offs(p0,168.03920000000002,274.86240000000004, 0), v100, z5, tool0;
MoveL Offs(p0,167.0625,274.8125, 0), v100, z5, tool0;
MoveL Offs(p0,166.14880000000002,275.08959999999996, 0), v100, z5, tool0;
MoveL Offs(p0,165.25189999999998,275.70029999999997, 0), v100, z5, tool0;
MoveL Offs(p0,164.3256,276.6512, 0), v100, z5, tool0;
MoveL Offs(p0,163.3237,277.9489, 0), v100, z5, tool0;
MoveL Offs(p0,162.2,279.6, 0), v100, z5, tool0;
MoveL Offs(p0,161.51600000000002,280.69220000000007, 0), v100, z5, tool0;
MoveL Offs(p0,160.96400000000006,281.68960000000004, 0), v100, z5, tool0;
MoveL Offs(p0,160.544,282.59340000000003, 0), v100, z5, tool0;
MoveL Offs(p0,160.25600000000003,283.4048000000001, 0), v100, z5, tool0;
MoveL Offs(p0,160.1,284.125, 0), v100, z5, tool0;
MoveL Offs(p0,160.076,284.75519999999995, 0), v100, z5, tool0;
MoveL Offs(p0,160.18399999999997,285.2966, 0), v100, z5, tool0;
MoveL Offs(p0,160.42400000000004,285.7504, 0), v100, z5, tool0;
MoveL Offs(p0,160.796,286.1178, 0), v100, z5, tool0;
MoveL Offs(p0,161.3,286.4, 0), v100, z5, tool0;
MoveL Offs(p0,162.04480000000007,286.62800000000004, 0), v100, z5, tool0;
MoveL Offs(p0,162.4862,286.67449999999997, 0), v100, z5, tool0;
MoveL Offs(p0,163.05840000000003,286.66400000000004, 0), v100, z5, tool0;
MoveL Offs(p0,167.92720000000003,285.872, 0), v100, z5, tool0;
MoveL Offs(p0,170.1074,285.4415, 0), v100, z5, tool0;
MoveL Offs(p0,172.8,284.9, 0), v100, z5, tool0;
MoveL Offs(p0,172.8,284.9, 0), v100, z5, tool0;
MoveJ Offs(p0,72.9,283.8, 10), v100, z1, tool0;
MoveL Offs(p0,74.3,281.6, 0), v100, z5, tool0;
MoveL Offs(p0,76.0,283.8, 0), v100, z5, tool0;
MoveL Offs(p0,76.63040000000001,284.55510000000004, 0), v100, z5, tool0;
MoveL Offs(p0,77.15520000000001,285.13680000000005, 0), v100, z5, tool0;
MoveL Offs(p0,77.59479999999999,285.5397, 0), v100, z5, tool0;
MoveL Offs(p0,77.9696,285.75840000000005, 0), v100, z5, tool0;
MoveL Offs(p0,78.3,285.7875, 0), v100, z5, tool0;
MoveL Offs(p0,78.6064,285.62160000000006, 0), v100, z5, tool0;
MoveL Offs(p0,78.9092,285.2553, 0), v100, z5, tool0;
MoveL Offs(p0,79.2288,284.68320000000006, 0), v100, z5, tool0;
MoveL Offs(p0,80.0,282.9, 0), v100, z5, tool0;
MoveL Offs(p0,80.24570000000001,282.3602, 0), v100, z5, tool0;
MoveL Offs(p0,80.50160000000002,281.88160000000005, 0), v100, z5, tool0;
MoveL Offs(p0,80.7659,281.4654, 0), v100, z5, tool0;
MoveL Offs(p0,81.0368,281.1128, 0), v100, z5, tool0;
MoveL Offs(p0,81.3125,280.825, 0), v100, z5, tool0;
MoveL Offs(p0,81.5912,280.60319999999996, 0), v100, z5, tool0;
MoveL Offs(p0,81.8711,280.4486, 0), v100, z5, tool0;
MoveL Offs(p0,82.15040000000002,280.36240000000004, 0), v100, z5, tool0;
MoveL Offs(p0,82.4273,280.3458, 0), v100, z5, tool0;
MoveL Offs(p0,82.7,280.4, 0), v100, z5, tool0;
MoveL Offs(p0,83.77099999999999,280.10810000000004, 0), v100, z5, tool0;
MoveL Offs(p0,83.756,279.86240000000004, 0), v100, z5, tool0;
MoveL Offs(p0,83.699,279.5603, 0), v100, z5, tool0;
MoveL Offs(p0,83.6,279.2, 0), v100, z5, tool0;
MoveL Offs(p0,83.35360000000003,278.36, 0), v100, z5, tool0;
MoveL Offs(p0,83.1869,277.742, 0), v100, z5, tool0;
MoveL Offs(p0,82.99680000000001,277.01599999999996, 0), v100, z5, tool0;
MoveL Offs(p0,82.7875,276.2, 0), v100, z5, tool0;
MoveL Offs(p0,82.56320000000001,275.312, 0), v100, z5, tool0;
MoveL Offs(p0,82.32809999999999,274.37, 0), v100, z5, tool0;
MoveL Offs(p0,82.0864,273.392, 0), v100, z5, tool0;
MoveL Offs(p0,81.8423,272.396, 0), v100, z5, tool0;
MoveL Offs(p0,81.6,271.4, 0), v100, z5, tool0;
MoveL Offs(p0,80.50630000000001,267.51720000000006, 0), v100, z5, tool0;
MoveL Offs(p0,79.17440000000002,263.54560000000004, 0), v100, z5, tool0;
MoveL Offs(p0,77.6481,259.5704, 0), v100, z5, tool0;
MoveL Offs(p0,75.9712,255.67680000000001, 0), v100, z5, tool0;
MoveL Offs(p0,74.1875,251.95, 0), v100, z5, tool0;
MoveL Offs(p0,72.3408,248.4752, 0), v100, z5, tool0;
MoveL Offs(p0,70.4749,245.33759999999998, 0), v100, z5, tool0;
MoveL Offs(p0,68.6336,242.62240000000003, 0), v100, z5, tool0;
MoveL Offs(p0,66.8607,240.4148, 0), v100, z5, tool0;
MoveL Offs(p0,65.2,238.8, 0), v100, z5, tool0;
MoveL Offs(p0,64.84270000000001,238.50610000000006, 0), v100, z5, tool0;
MoveL Offs(p0,64.54960000000003,238.28480000000008, 0), v100, z5, tool0;
MoveL Offs(p0,64.3189,238.13669999999996, 0), v100, z5, tool0;
MoveL Offs(p0,64.14880000000001,238.06240000000003, 0), v100, z5, tool0;
MoveL Offs(p0,64.0375,238.0625, 0), v100, z5, tool0;
MoveL Offs(p0,63.9832,238.13760000000002, 0), v100, z5, tool0;
MoveL Offs(p0,63.9841,238.28830000000002, 0), v100, z5, tool0;
MoveL Offs(p0,64.0384,238.5152, 0), v100, z5, tool0;
MoveL Offs(p0,64.3,239.2, 0), v100, z5, tool0;
MoveL Offs(p0,65.02470000000001,241.92600000000002, 0), v100, z5, tool0;
MoveL Offs(p0,65.6336,245.72000000000008, 0), v100, z5, tool0;
MoveL Offs(p0,66.1189,250.30599999999998, 0), v100, z5, tool0;
MoveL Offs(p0,66.4728,255.408, 0), v100, z5, tool0;
MoveL Offs(p0,66.6875,260.75, 0), v100, z5, tool0;
MoveL Offs(p0,66.75519999999999,266.05600000000004, 0), v100, z5, tool0;
MoveL Offs(p0,66.66810000000001,271.05, 0), v100, z5, tool0;
MoveL Offs(p0,66.4184,275.456, 0), v100, z5, tool0;
MoveL Offs(p0,65.9983,278.99800000000005, 0), v100, z5, tool0;
MoveL Offs(p0,65.4,281.4, 0), v100, z5, tool0;
MoveL Offs(p0,65.17280000000001,282.0720000000001, 0), v100, z5, tool0;
MoveL Offs(p0,65.1147,282.327, 0), v100, z5, tool0;
MoveL Offs(p0,65.09440000000001,282.528, 0), v100, z5, tool0;
MoveL Offs(p0,65.1125,282.675, 0), v100, z5, tool0;
MoveL Offs(p0,65.1696,282.768, 0), v100, z5, tool0;
MoveL Offs(p0,65.8,282.6, 0), v100, z5, tool0;
MoveL Offs(p0,67.22560000000001,282.8736, 0), v100, z5, tool0;
MoveL Offs(p0,67.4863,283.0928, 0), v100, z5, tool0;
MoveL Offs(p0,67.73920000000001,283.3552, 0), v100, z5, tool0;
MoveL Offs(p0,67.9789,283.6584, 0), v100, z5, tool0;
MoveL Offs(p0,68.2,284.0, 0), v100, z5, tool0;
MoveL Offs(p0,68.67450000000001,284.69910000000004, 0), v100, z5, tool0;
MoveL Offs(p0,69.14000000000001,285.2368000000001, 0), v100, z5, tool0;
MoveL Offs(p0,69.59949999999999,285.6137, 0), v100, z5, tool0;
MoveL Offs(p0,70.05600000000001,285.83040000000005, 0), v100, z5, tool0;
MoveL Offs(p0,70.5125,285.8875, 0), v100, z5, tool0;
MoveL Offs(p0,70.972,285.78560000000004, 0), v100, z5, tool0;
MoveL Offs(p0,71.4375,285.52529999999996, 0), v100, z5, tool0;
MoveL Offs(p0,71.912,285.10720000000003, 0), v100, z5, tool0;
MoveL Offs(p0,72.3985,284.5319, 0), v100, z5, tool0;
MoveL Offs(p0,72.9,283.8, 0), v100, z5, tool0;
MoveL Offs(p0,72.9,283.8, 0), v100, z5, tool0;
MoveJ Offs(p0,307.5,280.8, 10), v100, z1, tool0;
MoveL Offs(p0,308.595,279.56160000000006, 0), v100, z5, tool0;
MoveL Offs(p0,309.9720000000001,277.6848000000001, 0), v100, z5, tool0;
MoveL Offs(p0,311.64899999999994,275.1372, 0), v100, z5, tool0;
MoveL Offs(p0,313.644,271.88640000000004, 0), v100, z5, tool0;
MoveL Offs(p0,315.975,267.9, 0), v100, z5, tool0;
MoveL Offs(p0,318.65999999999997,263.1456, 0), v100, z5, tool0;
MoveL Offs(p0,321.717,257.5908, 0), v100, z5, tool0;
MoveL Offs(p0,325.16400000000004,251.2032, 0), v100, z5, tool0;
MoveL Offs(p0,329.01900000000006,243.9504, 0), v100, z5, tool0;
MoveL Offs(p0,333.3,235.8, 0), v100, z5, tool0;
MoveL Offs(p0,334.5212,233.51550000000003, 0), v100, z5, tool0;
MoveL Offs(p0,335.9416000000001,230.90400000000008, 0), v100, z5, tool0;
MoveL Offs(p0,337.5264,228.02849999999998, 0), v100, z5, tool0;
MoveL Offs(p0,339.24080000000004,224.952, 0), v100, z5, tool0;
MoveL Offs(p0,341.05,221.7375, 0), v100, z5, tool0;
MoveL Offs(p0,342.9192,218.448, 0), v100, z5, tool0;
MoveL Offs(p0,344.81359999999995,215.14649999999997, 0), v100, z5, tool0;
MoveL Offs(p0,346.69840000000005,211.89600000000002, 0), v100, z5, tool0;
MoveL Offs(p0,348.53880000000004,208.75950000000003, 0), v100, z5, tool0;
MoveL Offs(p0,350.3,205.8, 0), v100, z5, tool0;
MoveL Offs(p0,354.86300000000006,198.18660000000003, 0), v100, z5, tool0;
MoveL Offs(p0,358.6400000000001,191.81280000000004, 0), v100, z5, tool0;
MoveL Offs(p0,361.70300000000003,186.5382, 0), v100, z5, tool0;
MoveL Offs(p0,364.124,182.22240000000002, 0), v100, z5, tool0;
MoveL Offs(p0,365.975,178.725, 0), v100, z5, tool0;
MoveL Offs(p0,367.328,175.9056, 0), v100, z5, tool0;
MoveL Offs(p0,368.255,173.6238, 0), v100, z5, tool0;
MoveL Offs(p0,368.8280000000001,171.73920000000004, 0), v100, z5, tool0;
MoveL Offs(p0,369.119,170.1114, 0), v100, z5, tool0;
MoveL Offs(p0,369.2,168.6, 0), v100, z5, tool0;
MoveL Offs(p0,368.65200000000016,164.14560000000003, 0), v100, z5, tool0;
MoveL Offs(p0,367.931,162.0894, 0), v100, z5, tool0;
MoveL Offs(p0,366.88000000000005,160.10880000000003, 0), v100, z5, tool0;
MoveL Offs(p0,365.475,158.175, 0), v100, z5, tool0;
MoveL Offs(p0,363.69199999999995,156.2592, 0), v100, z5, tool0;
MoveL Offs(p0,361.50699999999995,154.3326, 0), v100, z5, tool0;
MoveL Offs(p0,358.8960000000001,152.36640000000003, 0), v100, z5, tool0;
MoveL Offs(p0,355.83500000000004,150.33180000000002, 0), v100, z5, tool0;
MoveL Offs(p0,352.3,148.2, 0), v100, z5, tool0;
MoveL Offs(p0,347.05490000000003,145.2118, 0), v100, z5, tool0;
MoveL Offs(p0,341.8152000000001,142.39040000000006, 0), v100, z5, tool0;
MoveL Offs(p0,336.66429999999997,139.7706, 0), v100, z5, tool0;
MoveL Offs(p0,331.68559999999997,137.3872, 0), v100, z5, tool0;
MoveL Offs(p0,326.9625,135.275, 0), v100, z5, tool0;
MoveL Offs(p0,322.5784,133.46880000000002, 0), v100, z5, tool0;
MoveL Offs(p0,318.6166999999999,132.0034, 0), v100, z5, tool0;
MoveL Offs(p0,315.1608,130.9136, 0), v100, z5, tool0;
MoveL Offs(p0,312.2941,130.23420000000002, 0), v100, z5, tool0;
MoveL Offs(p0,310.1,130.0, 0), v100, z5, tool0;
MoveL Offs(p0,306.4000000000001,130.52000000000004, 0), v100, z5, tool0;
MoveL Offs(p0,304.72700000000003,131.37699999999998, 0), v100, z5, tool0;
MoveL Offs(p0,303.036,132.816, 0), v100, z5, tool0;
MoveL Offs(p0,301.225,134.975, 0), v100, z5, tool0;
MoveL Offs(p0,299.192,137.99200000000002, 0), v100, z5, tool0;
MoveL Offs(p0,296.835,142.005, 0), v100, z5, tool0;
MoveL Offs(p0,294.052,147.152, 0), v100, z5, tool0;
MoveL Offs(p0,290.74100000000004,153.571, 0), v100, z5, tool0;
MoveL Offs(p0,286.8,161.4, 0), v100, z5, tool0;
MoveL Offs(p0,284.6310000000001,165.68460000000002, 0), v100, z5, tool0;
MoveL Offs(p0,282.4680000000001,169.91280000000006, 0), v100, z5, tool0;
MoveL Offs(p0,280.347,174.0162, 0), v100, z5, tool0;
MoveL Offs(p0,278.30400000000003,177.9264, 0), v100, z5, tool0;
MoveL Offs(p0,276.375,181.575, 0), v100, z5, tool0;
MoveL Offs(p0,274.59599999999995,184.8936, 0), v100, z5, tool0;
MoveL Offs(p0,273.003,187.81380000000001, 0), v100, z5, tool0;
MoveL Offs(p0,271.632,190.26720000000003, 0), v100, z5, tool0;
MoveL Offs(p0,270.519,192.18540000000002, 0), v100, z5, tool0;
MoveL Offs(p0,269.7,193.5, 0), v100, z5, tool0;
MoveL Offs(p0,267.13020000000006,197.23580000000004, 0), v100, z5, tool0;
MoveL Offs(p0,264.33360000000005,201.17440000000008, 0), v100, z5, tool0;
MoveL Offs(p0,261.3894,205.2126, 0), v100, z5, tool0;
MoveL Offs(p0,258.3768,209.24720000000002, 0), v100, z5, tool0;
MoveL Offs(p0,255.375,213.175, 0), v100, z5, tool0;
MoveL Offs(p0,252.46319999999997,216.8928, 0), v100, z5, tool0;
MoveL Offs(p0,249.72060000000002,220.2974, 0), v100, z5, tool0;
MoveL Offs(p0,247.2264,223.28560000000002, 0), v100, z5, tool0;
MoveL Offs(p0,245.0598,225.7542, 0), v100, z5, tool0;
MoveL Offs(p0,243.3,227.6, 0), v100, z5, tool0;
MoveL Offs(p0,241.58530000000002,229.36960000000005, 0), v100, z5, tool0;
MoveL Offs(p0,240.0944000000001,231.0288000000001, 0), v100, z5, tool0;
MoveL Offs(p0,238.81709999999993,232.59320000000002, 0), v100, z5, tool0;
MoveL Offs(p0,237.74320000000003,234.07840000000004, 0), v100, z5, tool0;
MoveL Offs(p0,236.8625,235.5, 0), v100, z5, tool0;
MoveL Offs(p0,236.1648,236.87359999999998, 0), v100, z5, tool0;
MoveL Offs(p0,235.63989999999998,238.21480000000003, 0), v100, z5, tool0;
MoveL Offs(p0,235.27759999999998,239.53920000000002, 0), v100, z5, tool0;
MoveL Offs(p0,235.0677,240.86239999999998, 0), v100, z5, tool0;
MoveL Offs(p0,235.0,242.2, 0), v100, z5, tool0;
MoveL Offs(p0,235.48320000000004,245.44560000000007, 0), v100, z5, tool0;
MoveL Offs(p0,236.07279999999997,246.7774, 0), v100, z5, tool0;
MoveL Offs(p0,236.92160000000004,247.9328, 0), v100, z5, tool0;
MoveL Offs(p0,238.05,248.925, 0), v100, z5, tool0;
MoveL Offs(p0,239.47839999999997,249.7672, 0), v100, z5, tool0;
MoveL Offs(p0,241.22719999999998,250.4726, 0), v100, z5, tool0;
MoveL Offs(p0,243.31680000000006,251.0544, 0), v100, z5, tool0;
MoveL Offs(p0,245.76760000000004,251.52580000000003, 0), v100, z5, tool0;
MoveL Offs(p0,248.6,251.9, 0), v100, z5, tool0;
MoveL Offs(p0,250.40150000000003,252.1486, 0), v100, z5, tool0;
MoveL Offs(p0,252.05600000000004,252.42480000000006, 0), v100, z5, tool0;
MoveL Offs(p0,253.60849999999996,252.7442, 0), v100, z5, tool0;
MoveL Offs(p0,255.10400000000004,253.12240000000003, 0), v100, z5, tool0;
MoveL Offs(p0,256.5875,253.575, 0), v100, z5, tool0;
MoveL Offs(p0,258.104,254.11759999999998, 0), v100, z5, tool0;
MoveL Offs(p0,259.6985,254.76579999999998, 0), v100, z5, tool0;
MoveL Offs(p0,261.41600000000005,255.53519999999997, 0), v100, z5, tool0;
MoveL Offs(p0,263.30150000000003,256.4414, 0), v100, z5, tool0;
MoveL Offs(p0,265.4,257.5, 0), v100, z5, tool0;
MoveL Offs(p0,269.27260000000007,259.5711, 0), v100, z5, tool0;
MoveL Offs(p0,272.75280000000004,261.5408000000001, 0), v100, z5, tool0;
MoveL Offs(p0,275.8742,263.4337, 0), v100, z5, tool0;
MoveL Offs(p0,278.67040000000003,265.2744, 0), v100, z5, tool0;
MoveL Offs(p0,281.175,267.0875, 0), v100, z5, tool0;
MoveL Offs(p0,283.4216,268.89759999999995, 0), v100, z5, tool0;
MoveL Offs(p0,285.4438,270.72929999999997, 0), v100, z5, tool0;
MoveL Offs(p0,287.27520000000004,272.60720000000003, 0), v100, z5, tool0;
MoveL Offs(p0,288.9494,274.5559, 0), v100, z5, tool0;
MoveL Offs(p0,290.5,276.6, 0), v100, z5, tool0;
MoveL Offs(p0,291.84950000000003,278.45410000000004, 0), v100, z5, tool0;
MoveL Offs(p0,292.9920000000001,279.96080000000006, 0), v100, z5, tool0;
MoveL Offs(p0,293.9785,281.1567, 0), v100, z5, tool0;
MoveL Offs(p0,294.86,282.0784, 0), v100, z5, tool0;
MoveL Offs(p0,295.6875,282.7625, 0), v100, z5, tool0;
MoveL Offs(p0,296.512,283.2456, 0), v100, z5, tool0;
MoveL Offs(p0,297.3845,283.5643, 0), v100, z5, tool0;
MoveL Offs(p0,298.35600000000005,283.75520000000006, 0), v100, z5, tool0;
MoveL Offs(p0,299.4775,283.8549, 0), v100, z5, tool0;
MoveL Offs(p0,300.8,283.9, 0), v100, z5, tool0;
MoveL Offs(p0,303.432,283.5144, 0), v100, z5, tool0;
MoveL Offs(p0,304.075,283.25, 0), v100, z5, tool0;
MoveL Offs(p0,304.724,282.9136, 0), v100, z5, tool0;
MoveL Offs(p0,305.385,282.5028, 0), v100, z5, tool0;
MoveL Offs(p0,306.064,282.0152, 0), v100, z5, tool0;
MoveL Offs(p0,306.767,281.4484, 0), v100, z5, tool0;
MoveL Offs(p0,307.5,280.8, 0), v100, z5, tool0;
MoveL Offs(p0,307.5,280.8, 0), v100, z5, tool0;
MoveJ Offs(p0,289.1,281.3, 10), v100, z1, tool0;
MoveL Offs(p0,288.82189999999997,279.1508, 0), v100, z5, tool0;
MoveL Offs(p0,288.20079999999996,278.06160000000006, 0), v100, z5, tool0;
MoveL Offs(p0,287.3625,276.85, 0), v100, z5, tool0;
MoveL Offs(p0,286.3352,275.5544, 0), v100, z5, tool0;
MoveL Offs(p0,285.1471,274.21320000000003, 0), v100, z5, tool0;
MoveL Offs(p0,283.82640000000004,272.8648, 0), v100, z5, tool0;
MoveL Offs(p0,282.4013,271.5476, 0), v100, z5, tool0;
MoveL Offs(p0,280.9,270.3, 0), v100, z5, tool0;
MoveL Offs(p0,278.93860000000006,268.86100000000005, 0), v100, z5, tool0;
MoveL Offs(p0,276.66880000000003,267.34400000000005, 0), v100, z5, tool0;
MoveL Offs(p0,274.2022,265.809, 0), v100, z5, tool0;
MoveL Offs(p0,271.6504,264.31600000000003, 0), v100, z5, tool0;
MoveL Offs(p0,269.125,262.925, 0), v100, z5, tool0;
MoveL Offs(p0,266.73760000000004,261.696, 0), v100, z5, tool0;
MoveL Offs(p0,264.5998,260.68899999999996, 0), v100, z5, tool0;
MoveL Offs(p0,262.8232,259.96400000000006, 0), v100, z5, tool0;
MoveL Offs(p0,261.5194,259.581, 0), v100, z5, tool0;
MoveL Offs(p0,260.8,259.6, 0), v100, z5, tool0;
MoveL Offs(p0,260.3707,259.825, 0), v100, z5, tool0;
MoveL Offs(p0,260.27840000000003,259.84000000000003, 0), v100, z5, tool0;
MoveL Offs(p0,260.2125,259.825, 0), v100, z5, tool0;
MoveL Offs(p0,260.3,259.3, 0), v100, z5, tool0;
MoveL Offs(p0,259.54670000000004,257.92569999999995, 0), v100, z5, tool0;
MoveL Offs(p0,258.6664,257.47440000000006, 0), v100, z5, tool0;
MoveL Offs(p0,257.5125,257.0375, 0), v100, z5, tool0;
MoveL Offs(p0,256.1096,256.62160000000006, 0), v100, z5, tool0;
MoveL Offs(p0,254.48230000000004,256.2333, 0), v100, z5, tool0;
MoveL Offs(p0,252.65520000000006,255.87920000000003, 0), v100, z5, tool0;
MoveL Offs(p0,250.6529,255.5659, 0), v100, z5, tool0;
MoveL Offs(p0,248.5,255.3, 0), v100, z5, tool0;
MoveL Offs(p0,246.51760000000007,255.0768000000001, 0), v100, z5, tool0;
MoveL Offs(p0,245.5489,254.93819999999997, 0), v100, z5, tool0;
MoveL Offs(p0,244.6168,254.78640000000004, 0), v100, z5, tool0;
MoveL Offs(p0,243.7375,254.625, 0), v100, z5, tool0;
MoveL Offs(p0,242.9272,254.4576, 0), v100, z5, tool0;
MoveL Offs(p0,242.20209999999997,254.28779999999998, 0), v100, z5, tool0;
MoveL Offs(p0,241.57840000000002,254.1192, 0), v100, z5, tool0;
MoveL Offs(p0,241.07229999999998,253.9554, 0), v100, z5, tool0;
MoveL Offs(p0,240.7,253.8, 0), v100, z5, tool0;
MoveL Offs(p0,240.23710000000005,253.56480000000002, 0), v100, z5, tool0;
MoveL Offs(p0,239.86480000000006,253.40640000000008, 0), v100, z5, tool0;
MoveL Offs(p0,239.5777,253.33559999999997, 0), v100, z5, tool0;
MoveL Offs(p0,239.37040000000002,253.36319999999995, 0), v100, z5, tool0;
MoveL Offs(p0,239.2375,253.5, 0), v100, z5, tool0;
MoveL Offs(p0,239.17329999999998,254.1444, 0), v100, z5, tool0;
MoveL Offs(p0,239.2312,254.67360000000002, 0), v100, z5, tool0;
MoveL Offs(p0,239.34189999999998,255.35520000000002, 0), v100, z5, tool0;
MoveL Offs(p0,239.5,256.2, 0), v100, z5, tool0;
MoveL Offs(p0,239.81680000000006,257.41600000000005, 0), v100, z5, tool0;
MoveL Offs(p0,240.02470000000002,258.10350000000005, 0), v100, z5, tool0;
MoveL Offs(p0,240.2584,258.824, 0), v100, z5, tool0;
MoveL Offs(p0,240.5125,259.5625, 0), v100, z5, tool0;
MoveL Offs(p0,240.78159999999997,260.304, 0), v100, z5, tool0;
MoveL Offs(p0,241.0603,261.0335, 0), v100, z5, tool0;
MoveL Offs(p0,241.34320000000002,261.73600000000005, 0), v100, z5, tool0;
MoveL Offs(p0,241.62490000000003,262.3965, 0), v100, z5, tool0;
MoveL Offs(p0,241.9,263.0, 0), v100, z5, tool0;
MoveL Offs(p0,243.7,266.5, 0), v100, z5, tool0;
MoveL Offs(p0,253.1,266.8, 0), v100, z5, tool0;
MoveL Offs(p0,258.60800000000006,267.09360000000004, 0), v100, z5, tool0;
MoveL Offs(p0,260.6645,267.39939999999996, 0), v100, z5, tool0;
MoveL Offs(p0,262.364,267.8768, 0), v100, z5, tool0;
MoveL Offs(p0,263.7875,268.575, 0), v100, z5, tool0;
MoveL Offs(p0,265.01599999999996,269.54319999999996, 0), v100, z5, tool0;
MoveL Offs(p0,266.1305,270.8306, 0), v100, z5, tool0;
MoveL Offs(p0,267.21200000000005,272.48640000000006, 0), v100, z5, tool0;
MoveL Offs(p0,268.3415,274.5598, 0), v100, z5, tool0;
MoveL Offs(p0,269.6,277.1, 0), v100, z5, tool0;
MoveL Offs(p0,272.5,283.3, 0), v100, z5, tool0;
MoveL Offs(p0,280.4,282.7, 0), v100, z5, tool0;
MoveL Offs(p0,282.9080000000001,282.48720000000014, 0), v100, z5, tool0;
MoveL Offs(p0,284.081,282.3598, 0), v100, z5, tool0;
MoveL Offs(p0,285.17600000000004,282.2216, 0), v100, z5, tool0;
MoveL Offs(p0,286.175,282.075, 0), v100, z5, tool0;
MoveL Offs(p0,287.06000000000006,281.9224, 0), v100, z5, tool0;
MoveL Offs(p0,287.813,281.7662, 0), v100, z5, tool0;
MoveL Offs(p0,288.41600000000005,281.60880000000003, 0), v100, z5, tool0;
MoveL Offs(p0,288.851,281.45259999999996, 0), v100, z5, tool0;
MoveL Offs(p0,289.1,281.3, 0), v100, z5, tool0;
MoveL Offs(p0,289.1,281.3, 0), v100, z5, tool0;
MoveJ Offs(p0,191.6,280.7, 10), v100, z1, tool0;
MoveL Offs(p0,191.3624,279.0908, 0), v100, z5, tool0;
MoveL Offs(p0,190.93280000000001,278.3496, 0), v100, z5, tool0;
MoveL Offs(p0,190.4,277.6, 0), v100, z5, tool0;
MoveL Offs(p0,189.80720000000002,276.8984, 0), v100, z5, tool0;
MoveL Offs(p0,189.19760000000002,276.3012, 0), v100, z5, tool0;
MoveL Offs(p0,188.61440000000002,275.8648, 0), v100, z5, tool0;
MoveL Offs(p0,188.1008,275.6456, 0), v100, z5, tool0;
MoveL Offs(p0,187.7,275.7, 0), v100, z5, tool0;
MoveL Offs(p0,187.29770000000002,275.3679, 0), v100, z5, tool0;
MoveL Offs(p0,187.4,275.2, 0), v100, z5, tool0;
MoveL Offs(p0,186.28000000000006,272.6464000000001, 0), v100, z5, tool0;
MoveL Offs(p0,184.5875,270.6586, 0), v100, z5, tool0;
MoveL Offs(p0,182.40000000000003,268.4272, 0), v100, z5, tool0;
MoveL Offs(p0,179.9125,266.125, 0), v100, z5, tool0;
MoveL Offs(p0,177.32,263.9248, 0), v100, z5, tool0;
MoveL Offs(p0,174.81749999999997,261.99940000000004, 0), v100, z5, tool0;
MoveL Offs(p0,172.6,260.52160000000003, 0), v100, z5, tool0;
MoveL Offs(p0,170.8625,259.6642, 0), v100, z5, tool0;
MoveL Offs(p0,169.8,259.6, 0), v100, z5, tool0;
MoveL Offs(p0,169.0301,260.07579999999996, 0), v100, z5, tool0;
MoveL Offs(p0,168.23680000000004,260.6464000000001, 0), v100, z5, tool0;
MoveL Offs(p0,167.44469999999998,261.28659999999996, 0), v100, z5, tool0;
MoveL Offs(p0,166.6784,261.9712, 0), v100, z5, tool0;
MoveL Offs(p0,165.9625,262.675, 0), v100, z5, tool0;
MoveL Offs(p0,165.32160000000002,263.3728, 0), v100, z5, tool0;
MoveL Offs(p0,164.78029999999998,264.0394, 0), v100, z5, tool0;
MoveL Offs(p0,164.3632,264.6496, 0), v100, z5, tool0;
MoveL Offs(p0,164.0949,265.1782, 0), v100, z5, tool0;
MoveL Offs(p0,164.0,265.6, 0), v100, z5, tool0;
MoveL Offs(p0,164.29600000000008,266.17200000000014, 0), v100, z5, tool0;
MoveL Offs(p0,164.64799999999997,266.599, 0), v100, z5, tool0;
MoveL Offs(p0,165.12,267.104, 0), v100, z5, tool0;
MoveL Offs(p0,165.7,267.675, 0), v100, z5, tool0;
MoveL Offs(p0,166.376,268.3, 0), v100, z5, tool0;
MoveL Offs(p0,167.13600000000002,268.967, 0), v100, z5, tool0;
MoveL Offs(p0,167.96800000000002,269.66400000000004, 0), v100, z5, tool0;
MoveL Offs(p0,168.85999999999999,270.379, 0), v100, z5, tool0;
MoveL Offs(p0,169.8,271.1, 0), v100, z5, tool0;
MoveL Offs(p0,170.7596,271.8502, 0), v100, z5, tool0;
MoveL Offs(p0,171.76480000000004,272.6496000000001, 0), v100, z5, tool0;
MoveL Offs(p0,172.79519999999997,273.4814, 0), v100, z5, tool0;
MoveL Offs(p0,173.8304,274.32880000000006, 0), v100, z5, tool0;
MoveL Offs(p0,174.85,275.175, 0), v100, z5, tool0;
MoveL Offs(p0,175.83360000000002,276.0032, 0), v100, z5, tool0;
MoveL Offs(p0,176.76079999999996,276.7966, 0), v100, z5, tool0;
MoveL Offs(p0,177.6112,277.5384, 0), v100, z5, tool0;
MoveL Offs(p0,178.3644,278.2118, 0), v100, z5, tool0;
MoveL Offs(p0,179.0,278.8, 0), v100, z5, tool0;
MoveL Offs(p0,179.8691,279.5967, 0), v100, z5, tool0;
MoveL Offs(p0,180.63680000000005,280.2536000000001, 0), v100, z5, tool0;
MoveL Offs(p0,181.3337,280.78090000000003, 0), v100, z5, tool0;
MoveL Offs(p0,181.99040000000005,281.1888, 0), v100, z5, tool0;
MoveL Offs(p0,182.6375,281.4875, 0), v100, z5, tool0;
MoveL Offs(p0,183.3056,281.68719999999996, 0), v100, z5, tool0;
MoveL Offs(p0,184.0253,281.7981, 0), v100, z5, tool0;
MoveL Offs(p0,184.82720000000003,281.8304, 0), v100, z5, tool0;
MoveL Offs(p0,185.74190000000002,281.7943, 0), v100, z5, tool0;
MoveL Offs(p0,186.8,281.7, 0), v100, z5, tool0;
MoveL Offs(p0,188.83849999999998,281.40840000000003, 0), v100, z5, tool0;
MoveL Offs(p0,189.44,281.3048, 0), v100, z5, tool0;
MoveL Offs(p0,189.9875,281.2, 0), v100, z5, tool0;
MoveL Offs(p0,190.47199999999998,281.09520000000003, 0), v100, z5, tool0;
MoveL Offs(p0,190.8845,280.9916, 0), v100, z5, tool0;
MoveL Offs(p0,191.216,280.89040000000006, 0), v100, z5, tool0;
MoveL Offs(p0,191.4575,280.79280000000006, 0), v100, z5, tool0;
MoveL Offs(p0,191.6,280.7, 0), v100, z5, tool0;
MoveL Offs(p0,191.6,280.7, 0), v100, z5, tool0;
MoveJ Offs(p0,203.7,278.3, 10), v100, z1, tool0;
MoveL Offs(p0,205.70480000000006,277.9608000000001, 0), v100, z5, tool0;
MoveL Offs(p0,206.49719999999996,277.7312, 0), v100, z5, tool0;
MoveL Offs(p0,207.1864,277.43440000000004, 0), v100, z5, tool0;
MoveL Offs(p0,207.8,277.05, 0), v100, z5, tool0;
MoveL Offs(p0,208.3656,276.5576, 0), v100, z5, tool0;
MoveL Offs(p0,208.91079999999997,275.9368, 0), v100, z5, tool0;
MoveL Offs(p0,209.4632,275.16720000000004, 0), v100, z5, tool0;
MoveL Offs(p0,210.0504,274.2284, 0), v100, z5, tool0;
MoveL Offs(p0,210.7,273.1, 0), v100, z5, tool0;
MoveL Offs(p0,211.87360000000004,271.11670000000004, 0), v100, z5, tool0;
MoveL Offs(p0,213.10480000000007,269.1976000000001, 0), v100, z5, tool0;
MoveL Offs(p0,214.3792,267.3589, 0), v100, z5, tool0;
MoveL Offs(p0,215.6824,265.61680000000007, 0), v100, z5, tool0;
MoveL Offs(p0,217.0,263.9875, 0), v100, z5, tool0;
MoveL Offs(p0,218.31760000000003,262.4871999999999, 0), v100, z5, tool0;
MoveL Offs(p0,219.6208,261.1321, 0), v100, z5, tool0;
MoveL Offs(p0,220.89520000000002,259.9384, 0), v100, z5, tool0;
MoveL Offs(p0,222.12640000000002,258.9223, 0), v100, z5, tool0;
MoveL Offs(p0,223.3,258.1, 0), v100, z5, tool0;
MoveL Offs(p0,224.4641,257.46510000000006, 0), v100, z5, tool0;
MoveL Offs(p0,225.85680000000008,256.8368000000001, 0), v100, z5, tool0;
MoveL Offs(p0,227.38869999999997,256.23969999999997, 0), v100, z5, tool0;
MoveL Offs(p0,228.9704,255.69840000000005, 0), v100, z5, tool0;
MoveL Offs(p0,230.5125,255.2375, 0), v100, z5, tool0;
MoveL Offs(p0,231.92560000000003,254.8816, 0), v100, z5, tool0;
MoveL Offs(p0,233.1203,254.65529999999998, 0), v100, z5, tool0;
MoveL Offs(p0,234.0072,254.58320000000003, 0), v100, z5, tool0;
MoveL Offs(p0,234.4969,254.68990000000002, 0), v100, z5, tool0;
MoveL Offs(p0,234.5,255.0, 0), v100, z5, tool0;
MoveL Offs(p0,234.71599999999998,255.8496, 0), v100, z5, tool0;
MoveL Offs(p0,234.87449999999998,255.99679999999998, 0), v100, z5, tool0;
MoveL Offs(p0,235.06000000000003,256.13919999999996, 0), v100, z5, tool0;
MoveL Offs(p0,235.26950000000002,256.2744, 0), v100, z5, tool0;
MoveL Offs(p0,235.5,256.4, 0), v100, z5, tool0;
MoveL Offs(p0,236.74020000000002,255.8339, 0), v100, z5, tool0;
MoveL Offs(p0,236.9384,255.25279999999998, 0), v100, z5, tool0;
MoveL Offs(p0,237.025,254.5625, 0), v100, z5, tool0;
MoveL Offs(p0,236.99759999999998,253.8152, 0), v100, z5, tool0;
MoveL Offs(p0,236.8538,253.0631, 0), v100, z5, tool0;
MoveL Offs(p0,236.59120000000001,252.35840000000002, 0), v100, z5, tool0;
MoveL Offs(p0,236.2074,251.75330000000002, 0), v100, z5, tool0;
MoveL Offs(p0,235.7,251.3, 0), v100, z5, tool0;
MoveL Offs(p0,234.6425,250.35070000000002, 0), v100, z5, tool0;
MoveL Offs(p0,233.75600000000009,248.99760000000006, 0), v100, z5, tool0;
MoveL Offs(p0,233.0495,247.32290000000003, 0), v100, z5, tool0;
MoveL Offs(p0,232.532,245.4088, 0), v100, z5, tool0;
MoveL Offs(p0,232.2125,243.3375, 0), v100, z5, tool0;
MoveL Offs(p0,232.1,241.19119999999998, 0), v100, z5, tool0;
MoveL Offs(p0,232.2035,239.05210000000002, 0), v100, z5, tool0;
MoveL Offs(p0,232.532,237.00240000000002, 0), v100, z5, tool0;
MoveL Offs(p0,233.0945,235.1243, 0), v100, z5, tool0;
MoveL Offs(p0,233.9,233.5, 0), v100, z5, tool0;
MoveL Offs(p0,234.2723,232.94829999999996, 0), v100, z5, tool0;
MoveL Offs(p0,234.77840000000006,232.26640000000006, 0), v100, z5, tool0;
MoveL Offs(p0,235.40210000000002,231.4741, 0), v100, z5, tool0;
MoveL Offs(p0,236.12720000000004,230.5912, 0), v100, z5, tool0;
MoveL Offs(p0,236.9375,229.6375, 0), v100, z5, tool0;
MoveL Offs(p0,237.81679999999997,228.6328, 0), v100, z5, tool0;
MoveL Offs(p0,238.7489,227.5969, 0), v100, z5, tool0;
MoveL Offs(p0,239.71760000000003,226.5496, 0), v100, z5, tool0;
MoveL Offs(p0,240.7067,225.51069999999999, 0), v100, z5, tool0;
MoveL Offs(p0,241.7,224.5, 0), v100, z5, tool0;
MoveL Offs(p0,243.94590000000002,222.18830000000003, 0), v100, z5, tool0;
MoveL Offs(p0,245.93920000000008,220.05840000000006, 0), v100, z5, tool0;
MoveL Offs(p0,247.67329999999998,218.11809999999997, 0), v100, z5, tool0;
MoveL Offs(p0,249.1416,216.37520000000004, 0), v100, z5, tool0;
MoveL Offs(p0,250.3375,214.8375, 0), v100, z5, tool0;
MoveL Offs(p0,251.25439999999998,213.51280000000003, 0), v100, z5, tool0;
MoveL Offs(p0,251.88569999999999,212.4089, 0), v100, z5, tool0;
MoveL Offs(p0,252.22480000000002,211.53360000000004, 0), v100, z5, tool0;
MoveL Offs(p0,252.2651,210.8947, 0), v100, z5, tool0;
MoveL Offs(p0,252.0,210.5, 0), v100, z5, tool0;
MoveL Offs(p0,251.42489999999998,210.2453, 0), v100, z5, tool0;
MoveL Offs(p0,251.22880000000004,210.2056, 0), v100, z5, tool0;
MoveL Offs(p0,251.0375,210.1875, 0), v100, z5, tool0;
MoveL Offs(p0,250.85520000000002,210.1904, 0), v100, z5, tool0;
MoveL Offs(p0,250.68609999999998,210.21370000000002, 0), v100, z5, tool0;
MoveL Offs(p0,250.5344,210.25680000000003, 0), v100, z5, tool0;
MoveL Offs(p0,250.53040000000001,210.96639999999996, 0), v100, z5, tool0;
MoveL Offs(p0,250.7023,210.9913, 0), v100, z5, tool0;
MoveL Offs(p0,250.9,211.0, 0), v100, z5, tool0;
MoveL Offs(p0,251.5,211.208, 0), v100, z5, tool0;
MoveL Offs(p0,251.575,211.3125, 0), v100, z5, tool0;
MoveL Offs(p0,251.61999999999998,211.43199999999996, 0), v100, z5, tool0;
MoveL Offs(p0,251.63500000000005,211.56350000000003, 0), v100, z5, tool0;
MoveL Offs(p0,251.62000000000003,211.704, 0), v100, z5, tool0;
MoveL Offs(p0,251.575,211.8505, 0), v100, z5, tool0;
MoveL Offs(p0,251.5,212.0, 0), v100, z5, tool0;
MoveL Offs(p0,251.17440000000005,212.37280000000004, 0), v100, z5, tool0;
MoveL Offs(p0,250.9906,212.4797, 0), v100, z5, tool0;
MoveL Offs(p0,250.79119999999998,212.5344, 0), v100, z5, tool0;
MoveL Offs(p0,250.575,212.5375, 0), v100, z5, tool0;
MoveL Offs(p0,250.3408,212.48960000000002, 0), v100, z5, tool0;
MoveL Offs(p0,250.08740000000003,212.3913, 0), v100, z5, tool0;
MoveL Offs(p0,249.81360000000004,212.24319999999997, 0), v100, z5, tool0;
MoveL Offs(p0,249.2,211.8, 0), v100, z5, tool0;
MoveL Offs(p0,248.84589999999997,211.48230000000004, 0), v100, z5, tool0;
MoveL Offs(p0,248.56320000000005,211.25040000000004, 0), v100, z5, tool0;
MoveL Offs(p0,248.35129999999998,211.10609999999997, 0), v100, z5, tool0;
MoveL Offs(p0,248.2096,211.05120000000002, 0), v100, z5, tool0;
MoveL Offs(p0,248.1375,211.0875, 0), v100, z5, tool0;
MoveL Offs(p0,248.1344,211.21679999999998, 0), v100, z5, tool0;
MoveL Offs(p0,248.19970000000004,211.4409, 0), v100, z5, tool0;
MoveL Offs(p0,248.53310000000002,212.18069999999997, 0), v100, z5, tool0;
MoveL Offs(p0,248.8,212.7, 0), v100, z5, tool0;
MoveL Offs(p0,249.0667,213.22970000000004, 0), v100, z5, tool0;
MoveL Offs(p0,249.2656000000001,213.68560000000008, 0), v100, z5, tool0;
MoveL Offs(p0,249.3949,214.0779, 0), v100, z5, tool0;
MoveL Offs(p0,249.45280000000002,214.41680000000002, 0), v100, z5, tool0;
MoveL Offs(p0,249.4375,214.7125, 0), v100, z5, tool0;
MoveL Offs(p0,249.3472,214.9752, 0), v100, z5, tool0;
MoveL Offs(p0,249.18009999999998,215.21509999999998, 0), v100, z5, tool0;
MoveL Offs(p0,248.2,215.9, 0), v100, z5, tool0;
MoveL Offs(p0,247.52640000000005,216.22400000000007, 0), v100, z5, tool0;
MoveL Offs(p0,247.1461,216.35899999999998, 0), v100, z5, tool0;
MoveL Offs(p0,246.74720000000002,216.47600000000003, 0), v100, z5, tool0;
MoveL Offs(p0,246.3375,216.575, 0), v100, z5, tool0;
MoveL Offs(p0,245.92479999999995,216.65600000000003, 0), v100, z5, tool0;
MoveL Offs(p0,245.5169,216.719, 0), v100, z5, tool0;
MoveL Offs(p0,245.12160000000003,216.76400000000004, 0), v100, z5, tool0;
MoveL Offs(p0,244.7467,216.791, 0), v100, z5, tool0;
MoveL Offs(p0,244.4,216.8, 0), v100, z5, tool0;
MoveL Offs(p0,240.5899,217.07509999999996, 0), v100, z5, tool0;
MoveL Offs(p0,239.91360000000003,217.17440000000002, 0), v100, z5, tool0;
MoveL Offs(p0,239.24570000000003,217.2833, 0), v100, z5, tool0;
MoveL Offs(p0,238.6,217.4, 0), v100, z5, tool0;
MoveL Offs(p0,236.78480000000005,217.71840000000006, 0), v100, z5, tool0;
MoveL Offs(p0,236.16369999999998,217.79509999999996, 0), v100, z5, tool0;
MoveL Offs(p0,235.71840000000003,217.8112, 0), v100, z5, tool0;
MoveL Offs(p0,235.4375,217.7625, 0), v100, z5, tool0;
MoveL Offs(p0,235.3096,217.64479999999998, 0), v100, z5, tool0;
MoveL Offs(p0,235.46720000000005,217.18560000000002, 0), v100, z5, tool0;
MoveL Offs(p0,235.7299,216.8357, 0), v100, z5, tool0;
MoveL Offs(p0,236.1,216.4, 0), v100, z5, tool0;
MoveL Offs(p0,236.42390000000006,215.96410000000006, 0), v100, z5, tool0;
MoveL Offs(p0,236.67520000000007,215.61280000000005, 0), v100, z5, tool0;
MoveL Offs(p0,236.85330000000005,215.34069999999997, 0), v100, z5, tool0;
MoveL Offs(p0,236.9576,215.14240000000004, 0), v100, z5, tool0;
MoveL Offs(p0,236.9875,215.0125, 0), v100, z5, tool0;
MoveL Offs(p0,236.9424,214.9456, 0), v100, z5, tool0;
MoveL Offs(p0,236.82169999999996,214.93630000000002, 0), v100, z5, tool0;
MoveL Offs(p0,236.62480000000005,214.97920000000005, 0), v100, z5, tool0;
MoveL Offs(p0,236.35110000000003,215.06890000000004, 0), v100, z5, tool0;
MoveL Offs(p0,234.87370000000004,215.59550000000004, 0), v100, z5, tool0;
MoveL Offs(p0,233.8416000000001,215.9400000000001, 0), v100, z5, tool0;
MoveL Offs(p0,232.91389999999996,216.23049999999998, 0), v100, z5, tool0;
MoveL Offs(p0,232.10080000000002,216.46400000000003, 0), v100, z5, tool0;
MoveL Offs(p0,231.4125,216.6375, 0), v100, z5, tool0;
MoveL Offs(p0,230.85920000000002,216.748, 0), v100, z5, tool0;
MoveL Offs(p0,230.4511,216.79249999999996, 0), v100, z5, tool0;
MoveL Offs(p0,230.19840000000005,216.76800000000003, 0), v100, z5, tool0;
MoveL Offs(p0,230.11129999999997,216.6715, 0), v100, z5, tool0;
MoveL Offs(p0,230.2,216.5, 0), v100, z5, tool0;
MoveL Offs(p0,230.42499999999995,215.95549999999997, 0), v100, z5, tool0;
MoveL Offs(p0,230.44,215.74, 0), v100, z5, tool0;
MoveL Offs(p0,230.425,215.5125, 0), v100, z5, tool0;
MoveL Offs(p0,229.9,214.3, 0), v100, z5, tool0;
MoveL Offs(p0,229.46840000000003,213.86240000000004, 0), v100, z5, tool0;
MoveL Offs(p0,229.02720000000005,213.5112000000001, 0), v100, z5, tool0;
MoveL Offs(p0,228.59679999999997,213.24880000000002, 0), v100, z5, tool0;
MoveL Offs(p0,228.19760000000005,213.0776, 0), v100, z5, tool0;
MoveL Offs(p0,227.85,213.0, 0), v100, z5, tool0;
MoveL Offs(p0,227.57440000000003,213.01839999999999, 0), v100, z5, tool0;
MoveL Offs(p0,227.39120000000003,213.1352, 0), v100, z5, tool0;
MoveL Offs(p0,227.32080000000005,213.35280000000003, 0), v100, z5, tool0;
MoveL Offs(p0,227.38360000000003,213.6736, 0), v100, z5, tool0;
MoveL Offs(p0,227.6,214.1, 0), v100, z5, tool0;
MoveL Offs(p0,227.21989999999997,214.86929999999998, 0), v100, z5, tool0;
MoveL Offs(p0,226.98560000000003,214.87120000000004, 0), v100, z5, tool0;
MoveL Offs(p0,226.7117,214.84790000000004, 0), v100, z5, tool0;
MoveL Offs(p0,226.4,214.8, 0), v100, z5, tool0;
MoveL Offs(p0,225.52879999999996,214.5039, 0), v100, z5, tool0;
MoveL Offs(p0,225.29760000000002,214.3648, 0), v100, z5, tool0;
MoveL Offs(p0,225.1,214.2125, 0), v100, z5, tool0;
MoveL Offs(p0,224.9384,214.05120000000002, 0), v100, z5, tool0;
MoveL Offs(p0,224.8152,213.88509999999997, 0), v100, z5, tool0;
MoveL Offs(p0,224.73280000000005,213.71840000000003, 0), v100, z5, tool0;
MoveL Offs(p0,224.69359999999998,213.5553, 0), v100, z5, tool0;
MoveL Offs(p0,224.7,213.4, 0), v100, z5, tool0;
MoveL Offs(p0,224.49300000000002,212.93919999999997, 0), v100, z5, tool0;
MoveL Offs(p0,224.30800000000005,212.7904, 0), v100, z5, tool0;
MoveL Offs(p0,224.075,212.65, 0), v100, z5, tool0;
MoveL Offs(p0,223.8,212.52159999999998, 0), v100, z5, tool0;
MoveL Offs(p0,223.48900000000003,212.40879999999999, 0), v100, z5, tool0;
MoveL Offs(p0,223.14800000000005,212.3152, 0), v100, z5, tool0;
MoveL Offs(p0,222.783,212.24439999999998, 0), v100, z5, tool0;
MoveL Offs(p0,222.4,212.2, 0), v100, z5, tool0;
MoveL Offs(p0,221.0698,211.95879999999997, 0), v100, z5, tool0;
MoveL Offs(p0,220.61759999999998,211.81760000000003, 0), v100, z5, tool0;
MoveL Offs(p0,220.175,211.65, 0), v100, z5, tool0;
MoveL Offs(p0,219.75039999999998,211.45839999999998, 0), v100, z5, tool0;
MoveL Offs(p0,219.35219999999998,211.2452, 0), v100, z5, tool0;
MoveL Offs(p0,218.9888,211.01280000000003, 0), v100, z5, tool0;
MoveL Offs(p0,218.66860000000003,210.76360000000005, 0), v100, z5, tool0;
MoveL Offs(p0,218.4,210.5, 0), v100, z5, tool0;
MoveL Offs(p0,217.83140000000003,210.01180000000005, 0), v100, z5, tool0;
MoveL Offs(p0,217.25920000000005,209.69040000000004, 0), v100, z5, tool0;
MoveL Offs(p0,216.67379999999997,209.54059999999998, 0), v100, z5, tool0;
MoveL Offs(p0,216.0656,209.56720000000004, 0), v100, z5, tool0;
MoveL Offs(p0,215.425,209.775, 0), v100, z5, tool0;
MoveL Offs(p0,214.7424,210.16879999999998, 0), v100, z5, tool0;
MoveL Offs(p0,214.0082,210.75339999999997, 0), v100, z5, tool0;
MoveL Offs(p0,213.21279999999996,211.53360000000004, 0), v100, z5, tool0;
MoveL Offs(p0,212.34660000000002,212.51420000000002, 0), v100, z5, tool0;
MoveL Offs(p0,211.4,213.7, 0), v100, z5, tool0;
MoveL Offs(p0,210.69740000000007,214.64990000000006, 0), v100, z5, tool0;
MoveL Offs(p0,210.14720000000003,215.41920000000005, 0), v100, z5, tool0;
MoveL Offs(p0,209.7458,216.03729999999996, 0), v100, z5, tool0;
MoveL Offs(p0,209.48959999999997,216.53360000000004, 0), v100, z5, tool0;
MoveL Offs(p0,209.375,216.9375, 0), v100, z5, tool0;
MoveL Offs(p0,209.39839999999998,217.2784, 0), v100, z5, tool0;
MoveL Offs(p0,209.5562,217.5857, 0), v100, z5, tool0;
MoveL Offs(p0,209.84480000000002,217.8888, 0), v100, z5, tool0;
MoveL Offs(p0,210.2606,218.21710000000002, 0), v100, z5, tool0;
MoveL Offs(p0,210.8,218.6, 0), v100, z5, tool0;
MoveL Offs(p0,212.40960000000004,219.77640000000002, 0), v100, z5, tool0;
MoveL Offs(p0,213.70480000000006,220.87120000000004, 0), v100, z5, tool0;
MoveL Offs(p0,214.69519999999997,221.9228, 0), v100, z5, tool0;
MoveL Offs(p0,215.3904,222.96960000000004, 0), v100, z5, tool0;
MoveL Offs(p0,215.8,224.05, 0), v100, z5, tool0;
MoveL Offs(p0,215.93359999999998,225.20239999999998, 0), v100, z5, tool0;
MoveL Offs(p0,215.80079999999998,226.4652, 0), v100, z5, tool0;
MoveL Offs(p0,215.4112,227.8768, 0), v100, z5, tool0;
MoveL Offs(p0,214.7744,229.4756, 0), v100, z5, tool0;
MoveL Offs(p0,213.9,231.3, 0), v100, z5, tool0;
MoveL Offs(p0,213.0863,232.84880000000004, 0), v100, z5, tool0;
MoveL Offs(p0,212.31040000000007,234.21040000000008, 0), v100, z5, tool0;
MoveL Offs(p0,211.5501,235.4076, 0), v100, z5, tool0;
MoveL Offs(p0,210.78320000000002,236.4632, 0), v100, z5, tool0;
MoveL Offs(p0,209.9875,237.4, 0), v100, z5, tool0;
MoveL Offs(p0,209.14080000000004,238.24079999999998, 0), v100, z5, tool0;
MoveL Offs(p0,208.22089999999997,239.0084, 0), v100, z5, tool0;
MoveL Offs(p0,207.2056,239.72560000000004, 0), v100, z5, tool0;
MoveL Offs(p0,206.0727,240.4152, 0), v100, z5, tool0;
MoveL Offs(p0,204.8,241.1, 0), v100, z5, tool0;
MoveL Offs(p0,203.28130000000004,241.7268, 0), v100, z5, tool0;
MoveL Offs(p0,201.49440000000007,242.2264000000001, 0), v100, z5, tool0;
MoveL Offs(p0,199.4531,242.59759999999997, 0), v100, z5, tool0;
MoveL Offs(p0,197.1712,242.83920000000003, 0), v100, z5, tool0;
MoveL Offs(p0,194.6625,242.95, 0), v100, z5, tool0;
MoveL Offs(p0,191.9408,242.9288, 0), v100, z5, tool0;
MoveL Offs(p0,189.01989999999998,242.7744, 0), v100, z5, tool0;
MoveL Offs(p0,185.91360000000003,242.48559999999998, 0), v100, z5, tool0;
MoveL Offs(p0,182.63569999999999,242.0612, 0), v100, z5, tool0;
MoveL Offs(p0,179.2,241.5, 0), v100, z5, tool0;
MoveL Offs(p0,176.9969,241.12270000000007, 0), v100, z5, tool0;
MoveL Offs(p0,175.20720000000006,240.83360000000008, 0), v100, z5, tool0;
MoveL Offs(p0,173.7703,240.63690000000003, 0), v100, z5, tool0;
MoveL Offs(p0,172.6256,240.53680000000003, 0), v100, z5, tool0;
MoveL Offs(p0,171.7125,240.5375, 0), v100, z5, tool0;
MoveL Offs(p0,170.97039999999998,240.64319999999998, 0), v100, z5, tool0;
MoveL Offs(p0,170.3387,240.85809999999998, 0), v100, z5, tool0;
MoveL Offs(p0,169.75680000000003,241.18640000000005, 0), v100, z5, tool0;
MoveL Offs(p0,168.5,242.2, 0), v100, z5, tool0;
MoveL Offs(p0,167.79670000000004,242.85930000000002, 0), v100, z5, tool0;
MoveL Offs(p0,167.19360000000003,243.50240000000002, 0), v100, z5, tool0;
MoveL Offs(p0,166.7009,244.1071, 0), v100, z5, tool0;
MoveL Offs(p0,166.3288,244.65120000000002, 0), v100, z5, tool0;
MoveL Offs(p0,166.0875,245.1125, 0), v100, z5, tool0;
MoveL Offs(p0,165.98719999999997,245.46880000000002, 0), v100, z5, tool0;
MoveL Offs(p0,166.0381,245.69790000000003, 0), v100, z5, tool0;
MoveL Offs(p0,166.2504,245.77760000000004, 0), v100, z5, tool0;
MoveL Offs(p0,166.6343,245.6857, 0), v100, z5, tool0;
MoveL Offs(p0,167.2,245.4, 0), v100, z5, tool0;
MoveL Offs(p0,167.67069999999998,245.18040000000002, 0), v100, z5, tool0;
MoveL Offs(p0,167.75840000000002,245.1728, 0), v100, z5, tool0;
MoveL Offs(p0,167.8125,245.2, 0), v100, z5, tool0;
MoveL Offs(p0,167.7049,245.6808, 0), v100, z5, tool0;
MoveL Offs(p0,167.6,245.9, 0), v100, z5, tool0;
MoveL Offs(p0,167.31760000000003,246.22160000000002, 0), v100, z5, tool0;
MoveL Offs(p0,167.1509,246.3509, 0), v100, z5, tool0;
MoveL Offs(p0,166.9728,246.45680000000002, 0), v100, z5, tool0;
MoveL Offs(p0,166.7875,246.5375, 0), v100, z5, tool0;
MoveL Offs(p0,166.59919999999997,246.59120000000001, 0), v100, z5, tool0;
MoveL Offs(p0,166.4121,246.61610000000002, 0), v100, z5, tool0;
MoveL Offs(p0,166.2304,246.61040000000003, 0), v100, z5, tool0;
MoveL Offs(p0,166.0583,246.57229999999998, 0), v100, z5, tool0;
MoveL Offs(p0,165.9,246.5, 0), v100, z5, tool0;
MoveL Offs(p0,165.4851,246.2453, 0), v100, z5, tool0;
MoveL Offs(p0,165.3672,246.2056, 0), v100, z5, tool0;
MoveL Offs(p0,165.2625,246.1875, 0), v100, z5, tool0;
MoveL Offs(p0,165.1728,246.1904, 0), v100, z5, tool0;
MoveL Offs(p0,165.0999,246.21369999999996, 0), v100, z5, tool0;
MoveL Offs(p0,165.0456,246.25680000000003, 0), v100, z5, tool0;
MoveL Offs(p0,164.7403,247.5746, 0), v100, z5, tool0;
MoveL Offs(p0,164.6672,247.81440000000003, 0), v100, z5, tool0;
MoveL Offs(p0,164.5869,248.0578, 0), v100, z5, tool0;
MoveL Offs(p0,164.5,248.3, 0), v100, z5, tool0;
MoveL Offs(p0,164.7799,249.37459999999996, 0), v100, z5, tool0;
MoveL Offs(p0,165.1528,249.84720000000002, 0), v100, z5, tool0;
MoveL Offs(p0,165.6625,250.375, 0), v100, z5, tool0;
MoveL Offs(p0,166.30720000000002,250.95680000000002, 0), v100, z5, tool0;
MoveL Offs(p0,167.0851,251.59140000000002, 0), v100, z5, tool0;
MoveL Offs(p0,167.9944,252.27760000000004, 0), v100, z5, tool0;
MoveL Offs(p0,169.0333,253.0142, 0), v100, z5, tool0;
MoveL Offs(p0,170.2,253.8, 0), v100, z5, tool0;
MoveL Offs(p0,172.58250000000004,255.46600000000004, 0), v100, z5, tool0;
MoveL Offs(p0,175.42400000000004,257.72, 0), v100, z5, tool0;
MoveL Offs(p0,178.5655,260.406, 0), v100, z5, tool0;
MoveL Offs(p0,181.848,263.36800000000005, 0), v100, z5, tool0;
MoveL Offs(p0,185.1125,266.45, 0), v100, z5, tool0;
MoveL Offs(p0,188.2,269.496, 0), v100, z5, tool0;
MoveL Offs(p0,190.95149999999998,272.35, 0), v100, z5, tool0;
MoveL Offs(p0,193.20800000000003,274.85600000000005, 0), v100, z5, tool0;
MoveL Offs(p0,194.8105,276.858, 0), v100, z5, tool0;
MoveL Offs(p0,195.6,278.2, 0), v100, z5, tool0;
MoveL Offs(p0,195.87680000000006,278.8728000000001, 0), v100, z5, tool0;
MoveL Offs(p0,196.0437,279.1297, 0), v100, z5, tool0;
MoveL Offs(p0,196.23040000000003,279.3344, 0), v100, z5, tool0;
MoveL Offs(p0,196.4375,279.4875, 0), v100, z5, tool0;
MoveL Offs(p0,196.6656,279.58959999999996, 0), v100, z5, tool0;
MoveL Offs(p0,196.9153,279.6413, 0), v100, z5, tool0;
MoveL Offs(p0,197.18720000000002,279.64320000000004, 0), v100, z5, tool0;
MoveL Offs(p0,197.4819,279.59590000000003, 0), v100, z5, tool0;
MoveL Offs(p0,197.8,279.5, 0), v100, z5, tool0;
MoveL Offs(p0,198.53840000000008,279.2888000000001, 0), v100, z5, tool0;
MoveL Offs(p0,199.03660000000002,279.16519999999997, 0), v100, z5, tool0;
MoveL Offs(p0,199.60320000000002,279.0344, 0), v100, z5, tool0;
MoveL Offs(p0,200.225,278.9, 0), v100, z5, tool0;
MoveL Offs(p0,200.8888,278.76559999999995, 0), v100, z5, tool0;
MoveL Offs(p0,201.58139999999997,278.6348, 0), v100, z5, tool0;
MoveL Offs(p0,202.2896,278.51120000000003, 0), v100, z5, tool0;
MoveL Offs(p0,203.0002,278.39840000000004, 0), v100, z5, tool0;
MoveL Offs(p0,203.7,278.3, 0), v100, z5, tool0;
MoveL Offs(p0,203.7,278.3, 0), v100, z5, tool0;
MoveJ Offs(p0,154.0,276.9, 10), v100, z1, tool0;
MoveL Offs(p0,154.2344,276.16330000000005, 0), v100, z5, tool0;
MoveL Offs(p0,154.87920000000003,274.8824000000001, 0), v100, z5, tool0;
MoveL Offs(p0,155.8468,273.19109999999995, 0), v100, z5, tool0;
MoveL Offs(p0,157.0496,271.2232, 0), v100, z5, tool0;
MoveL Offs(p0,158.4,269.1125, 0), v100, z5, tool0;
MoveL Offs(p0,159.81040000000002,266.9928, 0), v100, z5, tool0;
MoveL Offs(p0,161.1932,264.9979, 0), v100, z5, tool0;
MoveL Offs(p0,162.4608,263.2616, 0), v100, z5, tool0;
MoveL Offs(p0,163.5256,261.9177, 0), v100, z5, tool0;
MoveL Offs(p0,164.3,261.1, 0), v100, z5, tool0;
MoveL Offs(p0,164.9392,260.50120000000004, 0), v100, z5, tool0;
MoveL Offs(p0,165.41760000000005,259.8496000000001, 0), v100, z5, tool0;
MoveL Offs(p0,165.7364,259.15240000000006, 0), v100, z5, tool0;
MoveL Offs(p0,165.8968,258.4168, 0), v100, z5, tool0;
MoveL Offs(p0,165.9,257.65, 0), v100, z5, tool0;
MoveL Offs(p0,165.7472,256.8592, 0), v100, z5, tool0;
MoveL Offs(p0,165.43959999999998,256.05159999999995, 0), v100, z5, tool0;
MoveL Offs(p0,164.97840000000002,255.2344, 0), v100, z5, tool0;
MoveL Offs(p0,163.6,253.6, 0), v100, z5, tool0;
MoveL Offs(p0,162.67250000000004,252.6058, 0), v100, z5, tool0;
MoveL Offs(p0,161.92800000000005,251.7064000000001, 0), v100, z5, tool0;
MoveL Offs(p0,161.3635,250.8766, 0), v100, z5, tool0;
MoveL Offs(p0,160.97600000000003,250.09120000000001, 0), v100, z5, tool0;
MoveL Offs(p0,160.7625,249.325, 0), v100, z5, tool0;
MoveL Offs(p0,160.72000000000003,248.5528, 0), v100, z5, tool0;
MoveL Offs(p0,160.8455,247.74939999999998, 0), v100, z5, tool0;
MoveL Offs(p0,161.13600000000002,246.88960000000003, 0), v100, z5, tool0;
MoveL Offs(p0,161.5885,245.94819999999999, 0), v100, z5, tool0;
MoveL Offs(p0,162.2,244.9, 0), v100, z5, tool0;
MoveL Offs(p0,163.2373,243.09369999999998, 0), v100, z5, tool0;
MoveL Offs(p0,164.00640000000004,241.50160000000005, 0), v100, z5, tool0;
MoveL Offs(p0,164.50309999999996,240.10389999999998, 0), v100, z5, tool0;
MoveL Offs(p0,164.72320000000002,238.88080000000005, 0), v100, z5, tool0;
MoveL Offs(p0,164.6625,237.8125, 0), v100, z5, tool0;
MoveL Offs(p0,164.3168,236.8792, 0), v100, z5, tool0;
MoveL Offs(p0,163.68189999999998,236.06109999999998, 0), v100, z5, tool0;
MoveL Offs(p0,162.7536,235.3384, 0), v100, z5, tool0;
MoveL Offs(p0,161.5277,234.6913, 0), v100, z5, tool0;
MoveL Offs(p0,160.0,234.1, 0), v100, z5, tool0;
MoveL Offs(p0,159.0952,233.80720000000005, 0), v100, z5, tool0;
MoveL Offs(p0,158.34160000000003,233.59360000000007, 0), v100, z5, tool0;
MoveL Offs(p0,157.7104,233.46640000000002, 0), v100, z5, tool0;
MoveL Offs(p0,157.1728,233.43280000000004, 0), v100, z5, tool0;
MoveL Offs(p0,156.7,233.5, 0), v100, z5, tool0;
MoveL Offs(p0,156.2632,233.6752, 0), v100, z5, tool0;
MoveL Offs(p0,155.38240000000002,234.37840000000006, 0), v100, z5, tool0;
MoveL Offs(p0,154.88080000000002,234.9208, 0), v100, z5, tool0;
MoveL Offs(p0,154.3,235.6, 0), v100, z5, tool0;
MoveL Offs(p0,153.36380000000003,236.9368, 0), v100, z5, tool0;
MoveL Offs(p0,152.53440000000003,238.43440000000004, 0), v100, z5, tool0;
MoveL Offs(p0,151.8106,240.1036, 0), v100, z5, tool0;
MoveL Offs(p0,151.19120000000004,241.95520000000005, 0), v100, z5, tool0;
MoveL Offs(p0,150.675,244.0, 0), v100, z5, tool0;
MoveL Offs(p0,150.2608,246.2488, 0), v100, z5, tool0;
MoveL Offs(p0,149.9474,248.71240000000003, 0), v100, z5, tool0;
MoveL Offs(p0,149.73360000000002,251.40160000000006, 0), v100, z5, tool0;
MoveL Offs(p0,149.6182,254.3272, 0), v100, z5, tool0;
MoveL Offs(p0,149.6,257.5, 0), v100, z5, tool0;
MoveL Offs(p0,149.80080000000004,263.47200000000004, 0), v100, z5, tool0;
MoveL Offs(p0,150.03470000000002,266.33799999999997, 0), v100, z5, tool0;
MoveL Offs(p0,150.3424,269.03600000000006, 0), v100, z5, tool0;
MoveL Offs(p0,150.7125,271.5, 0), v100, z5, tool0;
MoveL Offs(p0,151.1336,273.66400000000004, 0), v100, z5, tool0;
MoveL Offs(p0,151.5943,275.462, 0), v100, z5, tool0;
MoveL Offs(p0,152.0832,276.82800000000003, 0), v100, z5, tool0;
MoveL Offs(p0,152.58890000000002,277.696, 0), v100, z5, tool0;
MoveL Offs(p0,153.1,278.0, 0), v100, z5, tool0;
MoveL Offs(p0,153.6328,277.78560000000004, 0), v100, z5, tool0;
MoveL Offs(p0,153.7375,277.675, 0), v100, z5, tool0;
MoveL Offs(p0,153.8272,277.5464, 0), v100, z5, tool0;
MoveL Offs(p0,153.9001,277.4022, 0), v100, z5, tool0;
MoveL Offs(p0,153.95440000000002,277.24480000000005, 0), v100, z5, tool0;
MoveL Offs(p0,153.9883,277.0766, 0), v100, z5, tool0;
MoveL Offs(p0,154.0,276.9, 0), v100, z5, tool0;
MoveL Offs(p0,154.0,276.9, 0), v100, z5, tool0;
MoveJ Offs(p0,229.5,269.4, 10), v100, z1, tool0;
MoveL Offs(p0,229.79570000000004,268.6701, 0), v100, z5, tool0;
MoveL Offs(p0,230.1376000000001,267.92880000000014, 0), v100, z5, tool0;
MoveL Offs(p0,230.5179,267.1887, 0), v100, z5, tool0;
MoveL Offs(p0,230.9288,266.4624, 0), v100, z5, tool0;
MoveL Offs(p0,231.3625,265.7625, 0), v100, z5, tool0;
MoveL Offs(p0,231.8112,265.1016, 0), v100, z5, tool0;
MoveL Offs(p0,232.26709999999997,264.4923, 0), v100, z5, tool0;
MoveL Offs(p0,232.72240000000002,263.9472, 0), v100, z5, tool0;
MoveL Offs(p0,233.16930000000002,263.4789, 0), v100, z5, tool0;
MoveL Offs(p0,233.6,263.1, 0), v100, z5, tool0;
MoveL Offs(p0,234.41000000000003,262.46360000000004, 0), v100, z5, tool0;
MoveL Offs(p0,235.0400000000001,261.92080000000004, 0), v100, z5, tool0;
MoveL Offs(p0,235.49,261.4512, 0), v100, z5, tool0;
MoveL Offs(p0,235.76000000000005,261.03440000000006, 0), v100, z5, tool0;
MoveL Offs(p0,235.85,260.65, 0), v100, z5, tool0;
MoveL Offs(p0,235.76,260.2776, 0), v100, z5, tool0;
MoveL Offs(p0,235.48999999999995,259.8968, 0), v100, z5, tool0;
MoveL Offs(p0,235.04000000000005,259.48720000000003, 0), v100, z5, tool0;
MoveL Offs(p0,234.41,259.02840000000003, 0), v100, z5, tool0;
MoveL Offs(p0,232.70610000000002,258.02000000000004, 0), v100, z5, tool0;
MoveL Offs(p0,231.76480000000006,257.7200000000001, 0), v100, z5, tool0;
MoveL Offs(p0,230.77669999999998,257.6, 0), v100, z5, tool0;
MoveL Offs(p0,229.7424,257.66, 0), v100, z5, tool0;
MoveL Offs(p0,228.6625,257.9, 0), v100, z5, tool0;
MoveL Offs(p0,226.3683,258.91999999999996, 0), v100, z5, tool0;
MoveL Offs(p0,225.1552,259.7, 0), v100, z5, tool0;
MoveL Offs(p0,223.8989,260.65999999999997, 0), v100, z5, tool0;
MoveL Offs(p0,222.6,261.8, 0), v100, z5, tool0;
MoveL Offs(p0,221.60220000000004,262.8292, 0), v100, z5, tool0;
MoveL Offs(p0,220.44960000000006,264.17760000000004, 0), v100, z5, tool0;
MoveL Offs(p0,219.20340000000002,265.7564, 0), v100, z5, tool0;
MoveL Offs(p0,217.9248,267.4768, 0), v100, z5, tool0;
MoveL Offs(p0,216.675,269.25, 0), v100, z5, tool0;
MoveL Offs(p0,215.5152,270.98720000000003, 0), v100, z5, tool0;
MoveL Offs(p0,214.5066,272.5996, 0), v100, z5, tool0;
MoveL Offs(p0,213.71040000000002,273.99840000000006, 0), v100, z5, tool0;
MoveL Offs(p0,213.1878,275.0948, 0), v100, z5, tool0;
MoveL Offs(p0,213.0,275.8, 0), v100, z5, tool0;
MoveL Offs(p0,213.37600000000006,276.0064000000001, 0), v100, z5, tool0;
MoveL Offs(p0,213.82349999999997,276.0421, 0), v100, z5, tool0;
MoveL Offs(p0,214.42400000000004,276.03520000000003, 0), v100, z5, tool0;
MoveL Offs(p0,219.19650000000001,275.42470000000003, 0), v100, z5, tool0;
MoveL Offs(p0,220.4,275.2, 0), v100, z5, tool0;
MoveL Offs(p0,227.8,273.8, 0), v100, z5, tool0;
MoveL Offs(p0,229.5,269.4, 0), v100, z5, tool0;
MoveL Offs(p0,229.5,269.4, 0), v100, z5, tool0;
MoveJ Offs(p0,334.1,248.3, 10), v100, z1, tool0;
MoveL Offs(p0,333.87750000000005,247.89480000000003, 0), v100, z5, tool0;
MoveL Offs(p0,333.6880000000001,247.57840000000004, 0), v100, z5, tool0;
MoveL Offs(p0,333.5285,247.3496, 0), v100, z5, tool0;
MoveL Offs(p0,333.396,247.20720000000006, 0), v100, z5, tool0;
MoveL Offs(p0,333.2875,247.15, 0), v100, z5, tool0;
MoveL Offs(p0,333.19999999999993,247.17680000000001, 0), v100, z5, tool0;
MoveL Offs(p0,333.13050000000004,247.28639999999996, 0), v100, z5, tool0;
MoveL Offs(p0,333.076,247.47760000000002, 0), v100, z5, tool0;
MoveL Offs(p0,333.0335,247.74920000000003, 0), v100, z5, tool0;
MoveL Offs(p0,333.0,248.1, 0), v100, z5, tool0;
MoveL Offs(p0,333.23760000000004,249.52199999999993, 0), v100, z5, tool0;
MoveL Offs(p0,333.4032,249.91600000000003, 0), v100, z5, tool0;
MoveL Offs(p0,333.6,250.25, 0), v100, z5, tool0;
MoveL Offs(p0,333.82079999999996,250.512, 0), v100, z5, tool0;
MoveL Offs(p0,334.0584,250.68999999999997, 0), v100, z5, tool0;
MoveL Offs(p0,334.3056,250.77200000000002, 0), v100, z5, tool0;
MoveL Offs(p0,334.55520000000007,250.746, 0), v100, z5, tool0;
MoveL Offs(p0,334.8,250.6, 0), v100, z5, tool0;
MoveL Offs(p0,334.5536,249.18110000000001, 0), v100, z5, tool0;
MoveL Offs(p0,334.42240000000004,248.89440000000005, 0), v100, z5, tool0;
MoveL Offs(p0,334.27080000000007,248.5993, 0), v100, z5, tool0;
MoveL Offs(p0,334.1,248.3, 0), v100, z5, tool0;
MoveL Offs(p0,334.1,248.3, 0), v100, z5, tool0;
MoveJ Offs(p0,365.5,243.9, 10), v100, z1, tool0;
MoveL Offs(p0,367.6965,242.47840000000002, 0), v100, z5, tool0;
MoveL Offs(p0,369.77600000000007,240.86720000000005, 0), v100, z5, tool0;
MoveL Offs(p0,371.7235,239.08679999999995, 0), v100, z5, tool0;
MoveL Offs(p0,373.52400000000006,237.1576, 0), v100, z5, tool0;
MoveL Offs(p0,375.1625,235.1, 0), v100, z5, tool0;
MoveL Offs(p0,376.62399999999997,232.93439999999995, 0), v100, z5, tool0;
MoveL Offs(p0,377.8935,230.6812, 0), v100, z5, tool0;
MoveL Offs(p0,378.956,228.3608, 0), v100, z5, tool0;
MoveL Offs(p0,379.79650000000004,225.99359999999996, 0), v100, z5, tool0;
MoveL Offs(p0,380.4,223.6, 0), v100, z5, tool0;
MoveL Offs(p0,381.19370000000004,220.45060000000004, 0), v100, z5, tool0;
MoveL Offs(p0,382.3216000000001,216.71680000000006, 0), v100, z5, tool0;
MoveL Offs(p0,383.70390000000003,212.60020000000003, 0), v100, z5, tool0;
MoveL Offs(p0,385.2608,208.30239999999998, 0), v100, z5, tool0;
MoveL Offs(p0,386.9125,204.025, 0), v100, z5, tool0;
MoveL Offs(p0,388.57919999999996,199.96959999999999, 0), v100, z5, tool0;
MoveL Offs(p0,390.1811,196.33780000000002, 0), v100, z5, tool0;
MoveL Offs(p0,391.63840000000005,193.33120000000002, 0), v100, z5, tool0;
MoveL Offs(p0,392.8713000000001,191.15140000000002, 0), v100, z5, tool0;
MoveL Offs(p0,393.8,190.0, 0), v100, z5, tool0;
MoveL Offs(p0,394.1736000000002,189.63920000000005, 0), v100, z5, tool0;
MoveL Offs(p0,394.4489,189.3358, 0), v100, z5, tool0;
MoveL Offs(p0,394.7728,188.9616, 0), v100, z5, tool0;
MoveL Offs(p0,395.1375,188.525, 0), v100, z5, tool0;
MoveL Offs(p0,395.5352,188.0344, 0), v100, z5, tool0;
MoveL Offs(p0,395.9581,187.4982, 0), v100, z5, tool0;
MoveL Offs(p0,396.39840000000004,186.9248, 0), v100, z5, tool0;
MoveL Offs(p0,396.8483,186.32260000000002, 0), v100, z5, tool0;
MoveL Offs(p0,397.3,185.7, 0), v100, z5, tool0;
MoveL Offs(p0,397.98190000000005,184.7846, 0), v100, z5, tool0;
MoveL Offs(p0,398.53120000000007,184.00480000000002, 0), v100, z5, tool0;
MoveL Offs(p0,398.95329999999996,183.34019999999998, 0), v100, z5, tool0;
MoveL Offs(p0,399.2536,182.7704, 0), v100, z5, tool0;
MoveL Offs(p0,399.4375,182.275, 0), v100, z5, tool0;
MoveL Offs(p0,399.5104,181.8336, 0), v100, z5, tool0;
MoveL Offs(p0,399.4777,181.42579999999998, 0), v100, z5, tool0;
MoveL Offs(p0,399.3448,181.03120000000004, 0), v100, z5, tool0;
MoveL Offs(p0,399.11710000000005,180.6294, 0), v100, z5, tool0;
MoveL Offs(p0,398.8,180.2, 0), v100, z5, tool0;
MoveL Offs(p0,398.4791000000001,179.792, 0), v100, z5, tool0;
MoveL Offs(p0,398.2368000000002,179.46800000000005, 0), v100, z5, tool0;
MoveL Offs(p0,398.0737,179.228, 0), v100, z5, tool0;
MoveL Offs(p0,397.9904,179.07199999999997, 0), v100, z5, tool0;
MoveL Offs(p0,397.9875,179.0, 0), v100, z5, tool0;
MoveL Offs(p0,398.0656,179.012, 0), v100, z5, tool0;
MoveL Offs(p0,398.22529999999995,179.108, 0), v100, z5, tool0;
MoveL Offs(p0,398.46720000000005,179.288, 0), v100, z5, tool0;
MoveL Offs(p0,399.2,179.9, 0), v100, z5, tool0;
MoveL Offs(p0,399.6323000000001,180.18980000000005, 0), v100, z5, tool0;
MoveL Offs(p0,400.0424000000001,180.39440000000005, 0), v100, z5, tool0;
MoveL Offs(p0,400.45009999999996,180.5066, 0), v100, z5, tool0;
MoveL Offs(p0,400.87520000000006,180.5192, 0), v100, z5, tool0;
MoveL Offs(p0,401.3375,180.425, 0), v100, z5, tool0;
MoveL Offs(p0,401.85679999999996,180.21679999999998, 0), v100, z5, tool0;
MoveL Offs(p0,403.14560000000006,179.42960000000002, 0), v100, z5, tool0;
MoveL Offs(p0,403.95470000000006,178.83620000000002, 0), v100, z5, tool0;
MoveL Offs(p0,404.9,178.1, 0), v100, z5, tool0;
MoveL Offs(p0,405.62260000000003,177.56220000000002, 0), v100, z5, tool0;
MoveL Offs(p0,406.4568000000001,176.97760000000005, 0), v100, z5, tool0;
MoveL Offs(p0,407.38219999999995,176.3594, 0), v100, z5, tool0;
MoveL Offs(p0,408.3784,175.72080000000003, 0), v100, z5, tool0;
MoveL Offs(p0,409.425,175.075, 0), v100, z5, tool0;
MoveL Offs(p0,410.50159999999994,174.4352, 0), v100, z5, tool0;
MoveL Offs(p0,411.58779999999996,173.8146, 0), v100, z5, tool0;
MoveL Offs(p0,412.6632000000001,173.2264, 0), v100, z5, tool0;
MoveL Offs(p0,413.70740000000006,172.68380000000002, 0), v100, z5, tool0;
MoveL Offs(p0,414.7,172.2, 0), v100, z5, tool0;
MoveL Offs(p0,416.1915000000001,171.54120000000003, 0), v100, z5, tool0;
MoveL Offs(p0,417.5360000000002,170.99760000000003, 0), v100, z5, tool0;
MoveL Offs(p0,418.8085,170.5584, 0), v100, z5, tool0;
MoveL Offs(p0,420.084,170.21280000000002, 0), v100, z5, tool0;
MoveL Offs(p0,421.4375,169.95, 0), v100, z5, tool0;
MoveL Offs(p0,422.9440000000001,169.7592, 0), v100, z5, tool0;
MoveL Offs(p0,424.6785,169.62959999999998, 0), v100, z5, tool0;
MoveL Offs(p0,426.716,169.55040000000002, 0), v100, z5, tool0;
MoveL Offs(p0,429.1315000000001,169.51080000000002, 0), v100, z5, tool0;
MoveL Offs(p0,432.0,169.5, 0), v100, z5, tool0;
MoveL Offs(p0,441.1360000000001,169.73680000000002, 0), v100, z5, tool0;
MoveL Offs(p0,442.625,169.925, 0), v100, z5, tool0;
MoveL Offs(p0,443.95200000000006,170.19119999999998, 0), v100, z5, tool0;
MoveL Offs(p0,445.195,170.5486, 0), v100, z5, tool0;
MoveL Offs(p0,446.43199999999996,171.01040000000003, 0), v100, z5, tool0;
MoveL Offs(p0,447.741,171.58980000000003, 0), v100, z5, tool0;
MoveL Offs(p0,449.2,172.3, 0), v100, z5, tool0;
MoveL Offs(p0,451.19410000000005,173.32530000000003, 0), v100, z5, tool0;
MoveL Offs(p0,452.9368000000001,174.32240000000007, 0), v100, z5, tool0;
MoveL Offs(p0,454.4587,175.3231, 0), v100, z5, tool0;
MoveL Offs(p0,455.7904,176.35920000000002, 0), v100, z5, tool0;
MoveL Offs(p0,456.9625,177.4625, 0), v100, z5, tool0;
MoveL Offs(p0,458.00559999999996,178.6648, 0), v100, z5, tool0;
MoveL Offs(p0,458.95029999999997,179.9979, 0), v100, z5, tool0;
MoveL Offs(p0,459.82720000000006,181.49360000000001, 0), v100, z5, tool0;
MoveL Offs(p0,460.6669,183.1837, 0), v100, z5, tool0;
MoveL Offs(p0,461.5,185.1, 0), v100, z5, tool0;
MoveL Offs(p0,462.06770000000006,186.50510000000003, 0), v100, z5, tool0;
MoveL Offs(p0,462.5136000000001,187.70080000000004, 0), v100, z5, tool0;
MoveL Offs(p0,462.8419,188.74769999999998, 0), v100, z5, tool0;
MoveL Offs(p0,463.0568,189.70639999999997, 0), v100, z5, tool0;
MoveL Offs(p0,463.1625,190.6375, 0), v100, z5, tool0;
MoveL Offs(p0,463.16319999999996,191.6016, 0), v100, z5, tool0;
MoveL Offs(p0,463.0631,192.65929999999997, 0), v100, z5, tool0;
MoveL Offs(p0,462.86640000000006,193.8712, 0), v100, z5, tool0;
MoveL Offs(p0,462.57730000000004,195.2979, 0), v100, z5, tool0;
MoveL Offs(p0,462.2,197.0, 0), v100, z5, tool0;
MoveL Offs(p0,461.71900000000016,198.78730000000002, 0), v100, z5, tool0;
MoveL Offs(p0,461.07600000000014,200.69040000000007, 0), v100, z5, tool0;
MoveL Offs(p0,460.30099999999993,202.65109999999999, 0), v100, z5, tool0;
MoveL Offs(p0,459.4240000000001,204.6112, 0), v100, z5, tool0;
MoveL Offs(p0,458.475,206.5125, 0), v100, z5, tool0;
MoveL Offs(p0,457.4839999999999,208.2968, 0), v100, z5, tool0;
MoveL Offs(p0,456.48100000000005,209.90590000000003, 0), v100, z5, tool0;
MoveL Offs(p0,455.496,211.28160000000003, 0), v100, z5, tool0;
MoveL Offs(p0,454.559,212.3657, 0), v100, z5, tool0;
MoveL Offs(p0,453.7,213.1, 0), v100, z5, tool0;
MoveL Offs(p0,453.44800000000004,213.38320000000007, 0), v100, z5, tool0;
MoveL Offs(p0,453.358,213.55180000000001, 0), v100, z5, tool0;
MoveL Offs(p0,453.2920000000001,213.73360000000002, 0), v100, z5, tool0;
MoveL Offs(p0,453.25,213.925, 0), v100, z5, tool0;
MoveL Offs(p0,453.23199999999997,214.12240000000003, 0), v100, z5, tool0;
MoveL Offs(p0,453.238,214.32219999999998, 0), v100, z5, tool0;
MoveL Offs(p0,453.26800000000003,214.52080000000007, 0), v100, z5, tool0;
MoveL Offs(p0,453.322,214.71459999999996, 0), v100, z5, tool0;
MoveL Offs(p0,453.4,214.9, 0), v100, z5, tool0;
MoveL Offs(p0,453.6492999999999,215.39950000000005, 0), v100, z5, tool0;
MoveL Offs(p0,453.68160000000006,215.54000000000002, 0), v100, z5, tool0;
MoveL Offs(p0,453.6875,215.6625, 0), v100, z5, tool0;
MoveL Offs(p0,453.66639999999995,215.76399999999998, 0), v100, z5, tool0;
MoveL Offs(p0,453.61769999999996,215.8415, 0), v100, z5, tool0;
MoveL Offs(p0,451.62700000000007,216.131, 0), v100, z5, tool0;
MoveL Offs(p0,451.3160000000001,216.23600000000002, 0), v100, z5, tool0;
MoveL Offs(p0,451.005,216.359, 0), v100, z5, tool0;
MoveL Offs(p0,450.7,216.5, 0), v100, z5, tool0;
MoveL Offs(p0,450.05120000000016,216.8136000000001, 0), v100, z5, tool0;
MoveL Offs(p0,449.82429999999994,216.98239999999996, 0), v100, z5, tool0;
MoveL Offs(p0,449.6616,217.16080000000002, 0), v100, z5, tool0;
MoveL Offs(p0,449.5625,217.35, 0), v100, z5, tool0;
MoveL Offs(p0,449.5263999999999,217.55119999999997, 0), v100, z5, tool0;
MoveL Offs(p0,449.5527,217.7656, 0), v100, z5, tool0;
MoveL Offs(p0,449.6408,217.99440000000004, 0), v100, z5, tool0;
MoveL Offs(p0,449.7901,218.2388, 0), v100, z5, tool0;
MoveL Offs(p0,450.0,218.5, 0), v100, z5, tool0;
MoveL Offs(p0,450.21590000000003,218.78560000000002, 0), v100, z5, tool0;
MoveL Offs(p0,450.3832000000001,219.04480000000007, 0), v100, z5, tool0;
MoveL Offs(p0,450.5012999999999,219.28119999999998, 0), v100, z5, tool0;
MoveL Offs(p0,450.5696,219.49840000000003, 0), v100, z5, tool0;
MoveL Offs(p0,450.5875,219.7, 0), v100, z5, tool0;
MoveL Offs(p0,450.5544,219.88959999999997, 0), v100, z5, tool0;
MoveL Offs(p0,450.4697,220.07079999999996, 0), v100, z5, tool0;
MoveL Offs(p0,450.33280000000013,220.24720000000002, 0), v100, z5, tool0;
MoveL Offs(p0,449.36359999999996,220.82229999999998, 0), v100, z5, tool0;
MoveL Offs(p0,449.26320000000004,220.83360000000002, 0), v100, z5, tool0;
MoveL Offs(p0,449.2,220.8125, 0), v100, z5, tool0;
MoveL Offs(p0,449.2952,220.39210000000003, 0), v100, z5, tool0;
MoveL Offs(p0,449.4,220.2, 0), v100, z5, tool0;
MoveL Offs(p0,449.649,219.746, 0), v100, z5, tool0;
MoveL Offs(p0,449.7720000000001,219.4120000000001, 0), v100, z5, tool0;
MoveL Offs(p0,449.733,219.20999999999998, 0), v100, z5, tool0;
MoveL Offs(p0,449.025,219.25, 0), v100, z5, tool0;
MoveL Offs(p0,448.284,219.516, 0), v100, z5, tool0;
MoveL Offs(p0,447.23699999999997,219.962, 0), v100, z5, tool0;
MoveL Offs(p0,445.84800000000007,220.6, 0), v100, z5, tool0;
MoveL Offs(p0,444.081,221.442, 0), v100, z5, tool0;
MoveL Offs(p0,441.9,222.5, 0), v100, z5, tool0;
MoveL Offs(p0,440.67980000000006,223.06840000000005, 0), v100, z5, tool0;
MoveL Offs(p0,439.4344000000001,223.62720000000007, 0), v100, z5, tool0;
MoveL Offs(p0,438.1866,224.16680000000002, 0), v100, z5, tool0;
MoveL Offs(p0,436.95920000000007,224.67759999999998, 0), v100, z5, tool0;
MoveL Offs(p0,435.775,225.15, 0), v100, z5, tool0;
MoveL Offs(p0,434.6567999999999,225.57440000000003, 0), v100, z5, tool0;
MoveL Offs(p0,433.62739999999997,225.94120000000004, 0), v100, z5, tool0;
